LIN {X 0,Y 452.247,Z 648.153,A -85,B 0,C 180,E1 20026.851,E2 20026.851} C_VEL
LIN {X 0,Y 448.409,Z 632.212,A -85,B 0,C 180,E1 20025.069,E2 20025.069} C_VEL
LIN {X 0,Y 446.45,Z 614.687,A -85,B 0,C 180,E1 20023.26,E2 20023.26} C_VEL
LIN {X 0,Y 446.584,Z 593.795,A -85,B 0,C 180,E1 20021.279,E2 20021.279} C_VEL
LIN {X 0,Y 452.628,Z 538.562,A -85,B 0,C 180,E1 20016.48,E2 20016.48} C_VEL
LIN {X 0,Y 452.905,Z 536.236,A -85,B 0,C 180,E1 20016.274,E2 20016.274} C_VEL
LIN {X 0,Y 443.763,Z 516.786,A -85,B 0,C 180,E1 20013.042,E2 20013.042} C_VEL
LIN {X 0,Y 435.011,Z 498.685,A -85,B 0,C 180,E1 20009.766,E2 20009.766} C_VEL
LIN {X 0,Y 426.568,Z 481.843,A -85,B 0,C 180,E1 20006.443,E2 20006.443} C_VEL
LIN {X 0,Y 421.16,Z 471.659,A -85,B 0,C 180,E1 20004.249,E2 20004.249} C_VEL
LIN {X 0,Y 419.437,Z 467.925,A -85,B 0,C 180,E1 20003.459,E2 20003.459} C_VEL
LIN {X 0,Y 417.555,Z 464.51,A -85,B 0,C 180,E1 20002.676,E2 20002.676} C_VEL
LIN {X 0,Y 417.359,Z 463.499,A -85,B 0,C 180,E1 20002.464,E2 20002.464} C_VEL
LIN {X 0,Y 417.347,Z 463.499,A -85,B 0,C 180,E1 19998.431,E2 19998.431} C_VEL
LIN {X 0,Y 417.376,Z 463.496,A -85,B 0,C 180,E1 19994.579,E2 19994.579} C_VEL
LIN {X 0,Y 417.334,Z 463.503,A -85,B 0,C 180,E1 19990.63,E2 19990.63} C_VEL
LIN {X 0,Y 417.38,Z 463.495,A -85,B 0,C 180,E1 19986.741,E2 19986.741} C_VEL
LIN {X 0,Y 417.352,Z 463.498,A -85,B 0,C 180,E1 19982.884,E2 19982.884} C_VEL
LIN {X 0,Y 417.382,Z 463.493,A -85,B 0,C 180,E1 19979.039,E2 19979.039} C_VEL
LIN {X 0,Y 417.345,Z 463.498,A -85,B 0,C 180,E1 19975.19,E2 19975.19} C_VEL
LIN {X 0,Y 417.377,Z 463.478,A -85,B 0,C 180,E1 19971.458,E2 19971.458} C_VEL
LIN {X 0,Y 417.342,Z 463.486,A -85,B 0,C 180,E1 19967.688,E2 19967.688} C_VEL
LIN {X 0,Y 417.362,Z 463.495,A -85,B 0,C 180,E1 19963.579,E2 19963.579} C_VEL
LIN {X 0,Y 417.369,Z 463.498,A -85,B 0,C 180,E1 19959.82,E2 19959.82} C_VEL
LIN {X 0,Y 417.363,Z 463.495,A -85,B 0,C 180,E1 19955.886,E2 19955.886} C_VEL
LIN {X 0,Y 417.385,Z 463.489,A -85,B 0,C 180,E1 19951.996,E2 19951.996} C_VEL
LIN {X 0,Y 417.38,Z 463.491,A -85,B 0,C 180,E1 19947.997,E2 19947.997} C_VEL
LIN {X 0,Y 417.367,Z 463.496,A -85,B 0,C 180,E1 19944.23,E2 19944.23} C_VEL
LIN {X 0,Y 417.349,Z 463.5,A -85,B 0,C 180,E1 19940.266,E2 19940.266} C_VEL
LIN {X 0,Y 417.374,Z 463.49,A -85,B 0,C 180,E1 19936.54,E2 19936.54} C_VEL
LIN {X 0,Y 417.39,Z 463.643,A -85,B 0,C 180,E1 19936.338,E2 19936.338} C_VEL
LIN {X 0,Y 418.712,Z 467.029,A -85,B 0,C 180,E1 19935.791,E2 19935.791} C_VEL
LIN {X 0,Y 419.888,Z 469.412,A -85,B 0,C 180,E1 19935.374,E2 19935.374} C_VEL
LIN {X 0,Y 426.66,Z 483.707,A -85,B 0,C 180,E1 19932.995,E2 19932.995} C_VEL
LIN {X 0,Y 433.872,Z 500.582,A -85,B 0,C 180,E1 19930.525,E2 19930.525} C_VEL
LIN {X 0,Y 444.251,Z 519.272,A -85,B 0,C 180,E1 19928.996,E2 19928.996} C_VEL
LIN {X 0,Y 445.887,Z 529.867,A -85,B 0,C 180,E1 19928.609,E2 19928.609} C_VEL
LIN {X 0,Y 439.801,Z 761.275,A -85,B 0,C 180,E1 19924.551,E2 19924.551} C_VEL
LIN {X 0,Y 438.683,Z 782.005,A -85,B 0,C 180,E1 19923.967,E2 19923.967} C_VEL
LIN {X 0,Y 437.32,Z 800.081,A -85,B 0,C 180,E1 19923.255,E2 19923.255} C_VEL
LIN {X 0,Y 435.806,Z 807.622,A -85,B 0,C 180,E1 19922.975,E2 19922.975} C_VEL
LIN {X 0,Y 429.22,Z 824.782,A -85,B 0,C 180,E1 19922.434,E2 19922.434} C_VEL
LIN {X 0,Y 427.352,Z 831.771,A -85,B 0,C 180,E1 19922.067,E2 19922.067} C_VEL
LIN {X 0,Y 427.21,Z 832.734,A -85,B 0,C 180,E1 19922,E2 19922} C_VEL
LIN {X 0,Y 424.828,Z 850.823,A -85,B 0,C 180,E1 19920.624,E2 19920.624} C_VEL
LIN {X 0,Y 422.226,Z 868.674,A -85,B 0,C 180,E1 19918.964,E2 19918.964} C_VEL
LIN {X 0,Y 419.559,Z 885.444,A -85,B 0,C 180,E1 19917.075,E2 19917.075} C_VEL
LIN {X 0,Y 417.031,Z 900.766,A -85,B 0,C 180,E1 19915.003,E2 19915.003} C_VEL
LIN {X 0,Y 414.786,Z 914.246,A -85,B 0,C 180,E1 19912.835,E2 19912.835} C_VEL
LIN {X 0,Y 412.756,Z 926.896,A -85,B 0,C 180,E1 19910.415,E2 19910.415} C_VEL
LIN {X 0,Y 411.086,Z 938.068,A -85,B 0,C 180,E1 19907.845,E2 19907.845} C_VEL
LIN {X 0,Y 409.863,Z 947.306,A -85,B 0,C 180,E1 19905.275,E2 19905.275} C_VEL
LIN {X 0,Y 408.984,Z 955.199,A -85,B 0,C 180,E1 19902.566,E2 19902.566} C_VEL
LIN {X 0,Y 408.421,Z 961.6,A -85,B 0,C 180,E1 19899.724,E2 19899.724} C_VEL
LIN {X 0,Y 408.141,Z 966.263,A -85,B 0,C 180,E1 19896.894,E2 19896.894} C_VEL
LIN {X 0,Y 408.022,Z 969.312,A -85,B 0,C 180,E1 19894.074,E2 19894.074} C_VEL
LIN {X 0,Y 407.98,Z 970.823,A -85,B 0,C 180,E1 19891.263,E2 19891.263} C_VEL
LIN {X 0,Y 407.98,Z 970.794,A -85,B 0,C 180,E1 19888.454,E2 19888.454} C_VEL
LIN {X 0,Y 408.024,Z 969.165,A -85,B 0,C 180,E1 19885.643,E2 19885.643} C_VEL
LIN {X 0,Y 408.152,Z 965.977,A -85,B 0,C 180,E1 19882.812,E2 19882.812} C_VEL
LIN {X 0,Y 408.449,Z 961.195,A -85,B 0,C 180,E1 19879.99,E2 19879.99} C_VEL
LIN {X 0,Y 409.002,Z 954.992,A -85,B 0,C 180,E1 19877.268,E2 19877.268} C_VEL
LIN {X 0,Y 409.947,Z 946.693,A -85,B 0,C 180,E1 19874.437,E2 19874.437} C_VEL
LIN {X 0,Y 411.285,Z 936.743,A -85,B 0,C 180,E1 19871.723,E2 19871.723} C_VEL
LIN {X 0,Y 412.905,Z 925.95,A -85,B 0,C 180,E1 19869.295,E2 19869.295} C_VEL
LIN {X 0,Y 414.977,Z 913.101,A -85,B 0,C 180,E1 19866.874,E2 19866.874} C_VEL
LIN {X 0,Y 417.417,Z 898.384,A -85,B 0,C 180,E1 19864.562,E2 19864.562} C_VEL
LIN {X 0,Y 420.016,Z 882.599,A -85,B 0,C 180,E1 19862.494,E2 19862.494} C_VEL
LIN {X 0,Y 422.519,Z 866.692,A -85,B 0,C 180,E1 19860.746,E2 19860.746} C_VEL
LIN {X 0,Y 425.074,Z 849.262,A -85,B 0,C 180,E1 19859.15,E2 19859.15} C_VEL
LIN {X 0,Y 427.469,Z 830.816,A -85,B 0,C 180,E1 19857.771,E2 19857.771} C_VEL
LIN {X 0,Y 429.58,Z 811.902,A -85,B 0,C 180,E1 19856.637,E2 19856.637} C_VEL
LIN {X 0,Y 431.357,Z 792.246,A -85,B 0,C 180,E1 19855.718,E2 19855.718} C_VEL
LIN {X 0,Y 432.78,Z 770.977,A -85,B 0,C 180,E1 19854.992,E2 19854.992} C_VEL
LIN {X 0,Y 433.737,Z 747.508,A -85,B 0,C 180,E1 19854.477,E2 19854.477} C_VEL
LIN {X 0,Y 439.275,Z 540.89,A -85,B 0,C 180,E1 19850.824,E2 19850.824} C_VEL
LIN {X 0,Y 433.898,Z 520.693,A -85,B 0,C 180,E1 19849.809,E2 19849.809} C_VEL
LIN {X 0,Y 423.787,Z 502.841,A -85,B 0,C 180,E1 19848.207,E2 19848.207} C_VEL
LIN {X 0,Y 418.624,Z 487.868,A -85,B 0,C 180,E1 19845.378,E2 19845.378} C_VEL
LIN {X 0,Y 413.554,Z 474.797,A -85,B 0,C 180,E1 19842.607,E2 19842.607} C_VEL
LIN {X 0,Y 410.381,Z 467.367,A -85,B 0,C 180,E1 19840.948,E2 19840.948} C_VEL
LIN {X 0,Y 410.03,Z 466.658,A -85,B 0,C 180,E1 19840.761,E2 19840.761} C_VEL
LIN {X 0,Y 415.308,Z 479.497,A -85,B 0,C 180,E1 19838.4,E2 19838.4} C_VEL
LIN {X 0,Y 422.076,Z 497.495,A -85,B 0,C 180,E1 19835.311,E2 19835.311} C_VEL
LIN {X 0,Y 428.337,Z 516.103,A -85,B 0,C 180,E1 19832.349,E2 19832.349} C_VEL
LIN {X 0,Y 425.447,Z 549.874,A -85,B 0,C 180,E1 19828.572,E2 19828.572} C_VEL
LIN {X 0,Y 422.614,Z 585.893,A -85,B 0,C 180,E1 19824.608,E2 19824.608} C_VEL
LIN {X 0,Y 420.128,Z 621.951,A -85,B 0,C 180,E1 19820.731,E2 19820.731} C_VEL
LIN {X 0,Y 420.828,Z 628.627,A -85,B 0,C 180,E1 19820.519,E2 19820.519} C_VEL
LIN {X 0,Y 416.374,Z 763.577,A -85,B 0,C 180,E1 19817.315,E2 19817.315} C_VEL
LIN {X 0,Y 415.988,Z 779.751,A -85,B 0,C 180,E1 19816.715,E2 19816.715} C_VEL
LIN {X 0,Y 415.353,Z 795.906,A -85,B 0,C 180,E1 19815.856,E2 19815.856} C_VEL
LIN {X 0,Y 414.592,Z 810.59,A -85,B 0,C 180,E1 19814.812,E2 19814.812} C_VEL
LIN {X 0,Y 413.68,Z 825.181,A -85,B 0,C 180,E1 19813.488,E2 19813.488} C_VEL
LIN {X 0,Y 412.722,Z 838.536,A -85,B 0,C 180,E1 19811.955,E2 19811.955} C_VEL
LIN {X 0,Y 411.812,Z 850.761,A -85,B 0,C 180,E1 19810.209,E2 19810.209} C_VEL
LIN {X 0,Y 410.995,Z 861.622,A -85,B 0,C 180,E1 19808.253,E2 19808.253} C_VEL
LIN {X 0,Y 410.392,Z 870.255,A -85,B 0,C 180,E1 19806.295,E2 19806.295} C_VEL
LIN {X 0,Y 409.918,Z 877.846,A -85,B 0,C 180,E1 19804.056,E2 19804.056} C_VEL
LIN {X 0,Y 409.653,Z 883.079,A -85,B 0,C 180,E1 19801.958,E2 19801.958} C_VEL
LIN {X 0,Y 409.548,Z 887.055,A -85,B 0,C 180,E1 19799.581,E2 19799.581} C_VEL
LIN {X 0,Y 409.583,Z 888.99,A -85,B 0,C 180,E1 19797.342,E2 19797.342} C_VEL
LIN {X 0,Y 409.775,Z 889.229,A -85,B 0,C 180,E1 19794.961,E2 19794.961} C_VEL
LIN {X 0,Y 410.11,Z 887.636,A -85,B 0,C 180,E1 19792.717,E2 19792.717} C_VEL
LIN {X 0,Y 410.655,Z 884.296,A -85,B 0,C 180,E1 19790.437,E2 19790.437} C_VEL
LIN {X 0,Y 411.479,Z 878.755,A -85,B 0,C 180,E1 19788.08,E2 19788.08} C_VEL
LIN {X 0,Y 412.372,Z 872.331,A -85,B 0,C 180,E1 19786.111,E2 19786.111} C_VEL
LIN {X 0,Y 413.597,Z 863.352,A -85,B 0,C 180,E1 19784.003,E2 19784.003} C_VEL
LIN {X 0,Y 414.895,Z 853.205,A -85,B 0,C 180,E1 19782.162,E2 19782.162} C_VEL
LIN {X 0,Y 416.186,Z 842.184,A -85,B 0,C 180,E1 19780.565,E2 19780.565} C_VEL
LIN {X 0,Y 417.51,Z 829.221,A -85,B 0,C 180,E1 19779.065,E2 19779.065} C_VEL
LIN {X 0,Y 418.633,Z 815.574,A -85,B 0,C 180,E1 19777.83,E2 19777.83} C_VEL
LIN {X 0,Y 419.575,Z 800.482,A -85,B 0,C 180,E1 19776.772,E2 19776.772} C_VEL
LIN {X 0,Y 420.221,Z 784.494,A -85,B 0,C 180,E1 19775.954,E2 19775.954} C_VEL
LIN {X 0,Y 421.597,Z 753.425,A -85,B 0,C 180,E1 19774.815,E2 19774.815} C_VEL
LIN {X 0,Y 431.426,Z 657.119,A -85,B 0,C 180,E1 19771.483,E2 19771.483} C_VEL
LIN {X 0,Y 438.558,Z 643.152,A -85,B 0,C 180,E1 19770.302,E2 19770.302} C_VEL
LIN {X 0,Y 445.715,Z 621.577,A -85,B 0,C 180,E1 19767.121,E2 19767.121} C_VEL
LIN {X 0,Y 453.266,Z 605.107,A -85,B 0,C 180,E1 19764.487,E2 19764.487} C_VEL
LIN {X 0,Y 461.57,Z 591.773,A -85,B 0,C 180,E1 19762.171,E2 19762.171} C_VEL
LIN {X 0,Y 453.703,Z 603.277,A -85,B 0,C 180,E1 19760.474,E2 19760.474} C_VEL
LIN {X 0,Y 447.749,Z 615.574,A -85,B 0,C 180,E1 19758.619,E2 19758.619} C_VEL
LIN {X 0,Y 444.305,Z 627.955,A -85,B 0,C 180,E1 19756.711,E2 19756.711} C_VEL
LIN {X 0,Y 443.385,Z 639.929,A -85,B 0,C 180,E1 19754.838,E2 19754.838} C_VEL
LIN {X 0,Y 444.836,Z 652.133,A -85,B 0,C 180,E1 19752.927,E2 19752.927} C_VEL
LIN {X 0,Y 448.588,Z 663.737,A -85,B 0,C 180,E1 19751.112,E2 19751.112} C_VEL
LIN {X 0,Y 454.843,Z 675.364,A -85,B 0,C 180,E1 19749.305,E2 19749.305} C_VEL
LIN {X 0,Y 461.889,Z 684.775,A -85,B 0,C 180,E1 19747.858,E2 19747.858} C_VEL
LIN {X 0,Y 450.972,Z 703.36,A -85,B 0,C 180,E1 19747.17,E2 19747.17} C_VEL
LIN {X 0,Y 442.545,Z 720.539,A -85,B 0,C 180,E1 19746.376,E2 19746.376} C_VEL
LIN {X 0,Y 438.274,Z 731,A -85,B 0,C 180,E1 19745.853,E2 19745.853} C_VEL
LIN {X 0,Y 435.008,Z 751.2,A -85,B 0,C 180,E1 19745.76,E2 19745.76} C_VEL
LIN {X 0,Y 432.722,Z 773.487,A -85,B 0,C 180,E1 19745.533,E2 19745.533} C_VEL
LIN {X 0,Y 431.639,Z 803.634,A -85,B 0,C 180,E1 19744.962,E2 19744.962} C_VEL
LIN {X 0,Y 430.206,Z 824.359,A -85,B 0,C 180,E1 19744.347,E2 19744.347} C_VEL
LIN {X 0,Y 428.359,Z 844.316,A -85,B 0,C 180,E1 19743.507,E2 19743.507} C_VEL
LIN {X 0,Y 426.167,Z 863.94,A -85,B 0,C 180,E1 19742.419,E2 19742.419} C_VEL
LIN {X 0,Y 423.795,Z 882.686,A -85,B 0,C 180,E1 19741.111,E2 19741.111} C_VEL
LIN {X 0,Y 421.195,Z 901.021,A -85,B 0,C 180,E1 19739.546,E2 19739.546} C_VEL
LIN {X 0,Y 418.667,Z 918.311,A -85,B 0,C 180,E1 19737.756,E2 19737.756} C_VEL
LIN {X 0,Y 416.222,Z 934.359,A -85,B 0,C 180,E1 19735.774,E2 19735.774} C_VEL
LIN {X 0,Y 414.071,Z 948.963,A -85,B 0,C 180,E1 19733.632,E2 19733.632} C_VEL
LIN {X 0,Y 412.098,Z 962.898,A -85,B 0,C 180,E1 19731.194,E2 19731.194} C_VEL
LIN {X 0,Y 410.508,Z 975.21,A -85,B 0,C 180,E1 19728.608,E2 19728.608} C_VEL
LIN {X 0,Y 409.439,Z 985.412,A -85,B 0,C 180,E1 19726.019,E2 19726.019} C_VEL
LIN {X 0,Y 408.7,Z 994.21,A -85,B 0,C 180,E1 19723.296,E2 19723.296} C_VEL
LIN {X 0,Y 408.279,Z 1001.508,A -85,B 0,C 180,E1 19720.442,E2 19720.442} C_VEL
LIN {X 0,Y 408.135,Z 1006.746,A -85,B 0,C 180,E1 19717.744,E2 19717.744} C_VEL
LIN {X 0,Y 408.111,Z 1010.345,A -85,B 0,C 180,E1 19715.061,E2 19715.061} C_VEL
LIN {X 0,Y 408.146,Z 1012.401,A -85,B 0,C 180,E1 19712.388,E2 19712.388} C_VEL
LIN {X 0,Y 408.157,Z 1012.992,A -85,B 0,C 180,E1 19709.58,E2 19709.58} C_VEL
LIN {X 0,Y 408.13,Z 1012.047,A -85,B 0,C 180,E1 19706.911,E2 19706.911} C_VEL
LIN {X 0,Y 408.1,Z 1009.523,A -85,B 0,C 180,E1 19704.236,E2 19704.236} C_VEL
LIN {X 0,Y 408.152,Z 1005.246,A -85,B 0,C 180,E1 19701.407,E2 19701.407} C_VEL
LIN {X 0,Y 408.354,Z 999.555,A -85,B 0,C 180,E1 19698.705,E2 19698.705} C_VEL
LIN {X 0,Y 408.82,Z 992.138,A -85,B 0,C 180,E1 19695.989,E2 19695.989} C_VEL
LIN {X 0,Y 409.665,Z 982.783,A -85,B 0,C 180,E1 19693.263,E2 19693.263} C_VEL
LIN {X 0,Y 410.881,Z 971.974,A -85,B 0,C 180,E1 19690.674,E2 19690.674} C_VEL
LIN {X 0,Y 412.492,Z 959.502,A -85,B 0,C 180,E1 19688.182,E2 19688.182} C_VEL
LIN {X 0,Y 414.56,Z 945.232,A -85,B 0,C 180,E1 19685.795,E2 19685.795} C_VEL
LIN {X 0,Y 416.83,Z 930.021,A -85,B 0,C 180,E1 19683.657,E2 19683.657} C_VEL
LIN {X 0,Y 419.242,Z 914.205,A -85,B 0,C 180,E1 19681.782,E2 19681.782} C_VEL
LIN {X 0,Y 421.803,Z 896.64,A -85,B 0,C 180,E1 19680.042,E2 19680.042} C_VEL
LIN {X 0,Y 424.332,Z 878.099,A -85,B 0,C 180,E1 19678.537,E2 19678.537} C_VEL
LIN {X 0,Y 426.655,Z 859.244,A -85,B 0,C 180,E1 19677.297,E2 19677.297} C_VEL
LIN {X 0,Y 428.718,Z 839.82,A -85,B 0,C 180,E1 19676.286,E2 19676.286} C_VEL
LIN {X 0,Y 430.514,Z 819.136,A -85,B 0,C 180,E1 19675.477,E2 19675.477} C_VEL
LIN {X 0,Y 431.819,Z 798.409,A -85,B 0,C 180,E1 19674.917,E2 19674.917} C_VEL
LIN {X 0,Y 432.958,Z 768.448,A -85,B 0,C 180,E1 19674.395,E2 19674.395} C_VEL
LIN {X 0,Y 434.942,Z 748.992,A -85,B 0,C 180,E1 19674.194,E2 19674.194} C_VEL
LIN {X 0,Y 448.015,Z 719.06,A -85,B 0,C 180,E1 19672.608,E2 19672.608} C_VEL
LIN {X 0,Y 457.258,Z 701.76,A -85,B 0,C 180,E1 19671.851,E2 19671.851} C_VEL
LIN {X 0,Y 465.342,Z 688.644,A -85,B 0,C 180,E1 19671.376,E2 19671.376} C_VEL
LIN {X 0,Y 456.514,Z 676.324,A -85,B 0,C 180,E1 19669.657,E2 19669.657} C_VEL
LIN {X 0,Y 449.449,Z 662.719,A -85,B 0,C 180,E1 19667.895,E2 19667.895} C_VEL
LIN {X 0,Y 444.221,Z 647.515,A -85,B 0,C 180,E1 19666.076,E2 19666.076} C_VEL
LIN {X 0,Y 440.778,Z 630.005,A -85,B 0,C 180,E1 19664.138,E2 19664.138} C_VEL
LIN {X 0,Y 439.519,Z 612.252,A -85,B 0,C 180,E1 19662.326,E2 19662.326} C_VEL
LIN {X 0,Y 440.316,Z 590.385,A -85,B 0,C 180,E1 19660.273,E2 19660.273} C_VEL
LIN {X 0,Y 445.999,Z 543.065,A -85,B 0,C 180,E1 19656.129,E2 19656.129} C_VEL
LIN {X 0,Y 446.371,Z 539.996,A -85,B 0,C 180,E1 19655.856,E2 19655.856} C_VEL
LIN {X 0,Y 436.422,Z 518.757,A -85,B 0,C 180,E1 19652.263,E2 19652.263} C_VEL
LIN {X 0,Y 427.384,Z 500.161,A -85,B 0,C 180,E1 19648.812,E2 19648.812} C_VEL
LIN {X 0,Y 418.385,Z 482.388,A -85,B 0,C 180,E1 19645.175,E2 19645.175} C_VEL
LIN {X 0,Y 413.379,Z 472.882,A -85,B 0,C 180,E1 19643.069,E2 19643.069} C_VEL
LIN {X 0,Y 411.325,Z 468.748,A -85,B 0,C 180,E1 19642.134,E2 19642.134} C_VEL
LIN {X 0,Y 409.559,Z 465.216,A -85,B 0,C 180,E1 19641.331,E2 19641.331} C_VEL
LIN {X 0,Y 409.423,Z 464.486,A -85,B 0,C 180,E1 19641.188,E2 19641.188} C_VEL
LIN {X 0,Y 409.427,Z 464.488,A -85,B 0,C 180,E1 19637.187,E2 19637.187} C_VEL
LIN {X 0,Y 409.442,Z 464.486,A -85,B 0,C 180,E1 19633.414,E2 19633.414} C_VEL
LIN {X 0,Y 409.438,Z 464.484,A -85,B 0,C 180,E1 19629.275,E2 19629.275} C_VEL
LIN {X 0,Y 409.427,Z 464.486,A -85,B 0,C 180,E1 19625.465,E2 19625.465} C_VEL
LIN {X 0,Y 409.435,Z 464.485,A -85,B 0,C 180,E1 19621.399,E2 19621.399} C_VEL
LIN {X 0,Y 409.423,Z 464.487,A -85,B 0,C 180,E1 19617.62,E2 19617.62} C_VEL
LIN {X 0,Y 409.404,Z 464.481,A -85,B 0,C 180,E1 19613.549,E2 19613.549} C_VEL
LIN {X 0,Y 409.434,Z 464.486,A -85,B 0,C 180,E1 19609.731,E2 19609.731} C_VEL
LIN {X 0,Y 409.393,Z 464.479,A -85,B 0,C 180,E1 19605.831,E2 19605.831} C_VEL
LIN {X 0,Y 409.437,Z 464.466,A -85,B 0,C 180,E1 19601.932,E2 19601.932} C_VEL
LIN {X 0,Y 409.419,Z 464.473,A -85,B 0,C 180,E1 19598.059,E2 19598.059} C_VEL
LIN {X 0,Y 409.442,Z 464.481,A -85,B 0,C 180,E1 19594.235,E2 19594.235} C_VEL
LIN {X 0,Y 409.413,Z 464.489,A -85,B 0,C 180,E1 19590.389,E2 19590.389} C_VEL
LIN {X 0,Y 409.442,Z 464.483,A -85,B 0,C 180,E1 19586.503,E2 19586.503} C_VEL
LIN {X 0,Y 409.404,Z 464.483,A -85,B 0,C 180,E1 19582.722,E2 19582.722} C_VEL
LIN {X 0,Y 409.416,Z 464.478,A -85,B 0,C 180,E1 19578.747,E2 19578.747} C_VEL
LIN {X 0,Y 409.454,Z 464.596,A -85,B 0,C 180,E1 19577.399,E2 19577.399} C_VEL
LIN {X 0,Y 410.728,Z 467.94,A -85,B 0,C 180,E1 19576.838,E2 19576.838} C_VEL
LIN {X 0,Y 411.906,Z 470.18,A -85,B 0,C 180,E1 19576.419,E2 19576.419} C_VEL
LIN {X 0,Y 418.963,Z 484.85,A -85,B 0,C 180,E1 19573.885,E2 19573.885} C_VEL
LIN {X 0,Y 426.18,Z 501.197,A -85,B 0,C 180,E1 19571.41,E2 19571.41} C_VEL
LIN {X 0,Y 438.347,Z 522.672,A -85,B 0,C 180,E1 19569.559,E2 19569.559} C_VEL
LIN {X 0,Y 439.628,Z 531.441,A -85,B 0,C 180,E1 19569.237,E2 19569.237} C_VEL
LIN {X 0,Y 433.238,Z 761.59,A -85,B 0,C 180,E1 19565.151,E2 19565.151} C_VEL
LIN {X 0,Y 432.073,Z 782.349,A -85,B 0,C 180,E1 19564.56,E2 19564.56} C_VEL
LIN {X 0,Y 430.416,Z 802.881,A -85,B 0,C 180,E1 19563.724,E2 19563.724} C_VEL
LIN {X 0,Y 428.44,Z 822.386,A -85,B 0,C 180,E1 19562.671,E2 19562.671} C_VEL
LIN {X 0,Y 427.21,Z 832.734,A -85,B 0,C 180,E1 19562,E2 19562} C_VEL
LIN {X 0,Y 425.5,Z 839.763,A -85,B 0,C 180,E1 19561.577,E2 19561.577} C_VEL
LIN {X 0,Y 417.937,Z 856.908,A -85,B 0,C 180,E1 19560.609,E2 19560.609} C_VEL
LIN {X 0,Y 416.078,Z 863.292,A -85,B 0,C 180,E1 19560.078,E2 19560.078} C_VEL
LIN {X 0,Y 413.363,Z 879.928,A -85,B 0,C 180,E1 19558.299,E2 19558.299} C_VEL
LIN {X 0,Y 410.686,Z 895.548,A -85,B 0,C 180,E1 19556.301,E2 19556.301} C_VEL
LIN {X 0,Y 408.214,Z 909.683,A -85,B 0,C 180,E1 19554.144,E2 19554.144} C_VEL
LIN {X 0,Y 405.949,Z 922.609,A -85,B 0,C 180,E1 19551.788,E2 19551.788} C_VEL
LIN {X 0,Y 404.098,Z 933.776,A -85,B 0,C 180,E1 19549.362,E2 19549.362} C_VEL
LIN {X 0,Y 402.506,Z 944.324,A -85,B 0,C 180,E1 19546.598,E2 19546.598} C_VEL
LIN {X 0,Y 401.402,Z 952.875,A -85,B 0,C 180,E1 19543.834,E2 19543.834} C_VEL
LIN {X 0,Y 400.688,Z 959.675,A -85,B 0,C 180,E1 19541.077,E2 19541.077} C_VEL
LIN {X 0,Y 400.274,Z 965.045,A -85,B 0,C 180,E1 19538.185,E2 19538.185} C_VEL
LIN {X 0,Y 400.068,Z 968.705,A -85,B 0,C 180,E1 19535.305,E2 19535.305} C_VEL
LIN {X 0,Y 400.006,Z 970.799,A -85,B 0,C 180,E1 19532.435,E2 19532.435} C_VEL
LIN {X 0,Y 399.991,Z 971.379,A -85,B 0,C 180,E1 19529.57,E2 19529.57} C_VEL
LIN {X 0,Y 400.015,Z 970.445,A -85,B 0,C 180,E1 19526.704,E2 19526.704} C_VEL
LIN {X 0,Y 400.115,Z 967.88,A -85,B 0,C 180,E1 19523.831,E2 19523.831} C_VEL
LIN {X 0,Y 400.362,Z 963.724,A -85,B 0,C 180,E1 19520.947,E2 19520.947} C_VEL
LIN {X 0,Y 400.847,Z 957.884,A -85,B 0,C 180,E1 19518.051,E2 19518.051} C_VEL
LIN {X 0,Y 401.675,Z 950.656,A -85,B 0,C 180,E1 19515.291,E2 19515.291} C_VEL
LIN {X 0,Y 402.918,Z 941.604,A -85,B 0,C 180,E1 19512.526,E2 19512.526} C_VEL
LIN {X 0,Y 404.663,Z 930.439,A -85,B 0,C 180,E1 19509.761,E2 19509.761} C_VEL
LIN {X 0,Y 406.836,Z 917.595,A -85,B 0,C 180,E1 19507.15,E2 19507.15} C_VEL
LIN {X 0,Y 409.221,Z 903.913,A -85,B 0,C 180,E1 19504.84,E2 19504.84} C_VEL
LIN {X 0,Y 411.772,Z 889.246,A -85,B 0,C 180,E1 19502.76,E2 19502.76} C_VEL
LIN {X 0,Y 414.527,Z 873.003,A -85,B 0,C 180,E1 19500.828,E2 19500.828} C_VEL
LIN {X 0,Y 417.337,Z 855.065,A -85,B 0,C 180,E1 19499.06,E2 19499.06} C_VEL
LIN {X 0,Y 419.924,Z 837.057,A -85,B 0,C 180,E1 19497.605,E2 19497.605} C_VEL
LIN {X 0,Y 422.208,Z 818.712,A -85,B 0,C 180,E1 19496.398,E2 19496.398} C_VEL
LIN {X 0,Y 424.212,Z 799.183,A -85,B 0,C 180,E1 19495.386,E2 19495.386} C_VEL
LIN {X 0,Y 425.793,Z 779.188,A -85,B 0,C 180,E1 19494.615,E2 19494.615} C_VEL
LIN {X 0,Y 426.869,Z 758.771,A -85,B 0,C 180,E1 19494.067,E2 19494.067} C_VEL
LIN {X 0,Y 433.03,Z 542.633,A -85,B 0,C 180,E1 19490.18,E2 19490.18} C_VEL
LIN {X 0,Y 428.346,Z 524.911,A -85,B 0,C 180,E1 19489.267,E2 19489.267} C_VEL
LIN {X 0,Y 417.742,Z 506.393,A -85,B 0,C 180,E1 19487.569,E2 19487.569} C_VEL
LIN {X 0,Y 416.036,Z 503.201,A -85,B 0,C 180,E1 19487.241,E2 19487.241} C_VEL
LIN {X 0,Y 410.685,Z 488.339,A -85,B 0,C 180,E1 19484.326,E2 19484.326} C_VEL
LIN {X 0,Y 405.937,Z 476.291,A -85,B 0,C 180,E1 19481.685,E2 19481.685} C_VEL
LIN {X 0,Y 404.161,Z 472.316,A -85,B 0,C 180,E1 19480.738,E2 19480.738} C_VEL
LIN {X 0,Y 411.069,Z 489.811,A -85,B 0,C 180,E1 19477.537,E2 19477.537} C_VEL
LIN {X 0,Y 417.829,Z 508.675,A -85,B 0,C 180,E1 19474.351,E2 19474.351} C_VEL
LIN {X 0,Y 421.262,Z 519.171,A -85,B 0,C 180,E1 19472.682,E2 19472.682} C_VEL
LIN {X 0,Y 418.161,Z 553.481,A -85,B 0,C 180,E1 19468.804,E2 19468.804} C_VEL
LIN {X 0,Y 415.231,Z 589.559,A -85,B 0,C 180,E1 19464.795,E2 19464.795} C_VEL
LIN {X 0,Y 412.862,Z 623.388,A -85,B 0,C 180,E1 19461.15,E2 19461.15} C_VEL
LIN {X 0,Y 413.48,Z 629.666,A -85,B 0,C 180,E1 19460.943,E2 19460.943} C_VEL
LIN {X 0,Y 408.78,Z 764.001,A -85,B 0,C 180,E1 19457.659,E2 19457.659} C_VEL
LIN {X 0,Y 408.388,Z 780.031,A -85,B 0,C 180,E1 19457.062,E2 19457.062} C_VEL
LIN {X 0,Y 407.703,Z 796.723,A -85,B 0,C 180,E1 19456.162,E2 19456.162} C_VEL
LIN {X 0,Y 406.907,Z 811.445,A -85,B 0,C 180,E1 19455.098,E2 19455.098} C_VEL
LIN {X 0,Y 405.936,Z 826.289,A -85,B 0,C 180,E1 19453.727,E2 19453.727} C_VEL
LIN {X 0,Y 404.953,Z 839.471,A -85,B 0,C 180,E1 19452.187,E2 19452.187} C_VEL
LIN {X 0,Y 404.002,Z 851.751,A -85,B 0,C 180,E1 19450.409,E2 19450.409} C_VEL
LIN {X 0,Y 403.146,Z 862.656,A -85,B 0,C 180,E1 19448.414,E2 19448.414} C_VEL
LIN {X 0,Y 402.516,Z 871.354,A -85,B 0,C 180,E1 19446.418,E2 19446.418} C_VEL
LIN {X 0,Y 402.022,Z 879.004,A -85,B 0,C 180,E1 19444.136,E2 19444.136} C_VEL
LIN {X 0,Y 401.749,Z 884.296,A -85,B 0,C 180,E1 19441.997,E2 19441.997} C_VEL
LIN {X 0,Y 401.644,Z 888.328,A -85,B 0,C 180,E1 19439.572,E2 19439.572} C_VEL
LIN {X 0,Y 401.692,Z 890.316,A -85,B 0,C 180,E1 19437.29,E2 19437.29} C_VEL
LIN {X 0,Y 401.909,Z 890.606,A -85,B 0,C 180,E1 19434.862,E2 19434.862} C_VEL
LIN {X 0,Y 402.286,Z 889.071,A -85,B 0,C 180,E1 19432.574,E2 19432.574} C_VEL
LIN {X 0,Y 402.877,Z 885.858,A -85,B 0,C 180,E1 19430.284,E2 19430.284} C_VEL
LIN {X 0,Y 403.719,Z 880.679,A -85,B 0,C 180,E1 19427.993,E2 19427.993} C_VEL
LIN {X 0,Y 404.763,Z 873.969,A -85,B 0,C 180,E1 19425.845,E2 19425.845} C_VEL
LIN {X 0,Y 405.994,Z 865.73,A -85,B 0,C 180,E1 19423.839,E2 19423.839} C_VEL
LIN {X 0,Y 407.358,Z 855.976,A -85,B 0,C 180,E1 19421.985,E2 19421.985} C_VEL
LIN {X 0,Y 408.83,Z 844.758,A -85,B 0,C 180,E1 19420.276,E2 19420.276} C_VEL
LIN {X 0,Y 410.28,Z 831.662,A -85,B 0,C 180,E1 19418.709,E2 19418.709} C_VEL
LIN {X 0,Y 411.54,Z 818.132,A -85,B 0,C 180,E1 19417.427,E2 19417.427} C_VEL
LIN {X 0,Y 412.561,Z 803.674,A -85,B 0,C 180,E1 19416.364,E2 19416.364} C_VEL
LIN {X 0,Y 413.348,Z 787.167,A -85,B 0,C 180,E1 19415.47,E2 19415.47} C_VEL
LIN {X 0,Y 414.903,Z 756.833,A -85,B 0,C 180,E1 19414.279,E2 19414.279} C_VEL
LIN {X 0,Y 425.848,Z 660.115,A -85,B 0,C 180,E1 19410.767,E2 19410.767} C_VEL
LIN {X 0,Y 433.367,Z 645.952,A -85,B 0,C 180,E1 19409.574,E2 19409.574} C_VEL
LIN {X 0,Y 441.041,Z 625.163,A -85,B 0,C 180,E1 19406.416,E2 19406.416} C_VEL
LIN {X 0,Y 449.009,Z 609.528,A -85,B 0,C 180,E1 19403.836,E2 19403.836} C_VEL
LIN {X 0,Y 454.853,Z 600.657,A -85,B 0,C 180,E1 19402.236,E2 19402.236} C_VEL
LIN {X 0,Y 447.156,Z 612.063,A -85,B 0,C 180,E1 19400.484,E2 19400.484} C_VEL
LIN {X 0,Y 441.777,Z 623.28,A -85,B 0,C 180,E1 19398.713,E2 19398.713} C_VEL
LIN {X 0,Y 438.509,Z 635.367,A -85,B 0,C 180,E1 19396.762,E2 19396.762} C_VEL
LIN {X 0,Y 437.725,Z 647.141,A -85,B 0,C 180,E1 19394.836,E2 19394.836} C_VEL
LIN {X 0,Y 439.408,Z 659.195,A -85,B 0,C 180,E1 19392.873,E2 19392.873} C_VEL
LIN {X 0,Y 443.526,Z 670.976,A -85,B 0,C 180,E1 19390.957,E2 19390.957} C_VEL
LIN {X 0,Y 449.983,Z 682.329,A -85,B 0,C 180,E1 19389.128,E2 19389.128} C_VEL
LIN {X 0,Y 453.361,Z 687.303,A -85,B 0,C 180,E1 19388.364,E2 19388.364} C_VEL
LIN {X 0,Y 442.963,Z 705.582,A -85,B 0,C 180,E1 19387.656,E2 19387.656} C_VEL
LIN {X 0,Y 434.5,Z 723.436,A -85,B 0,C 180,E1 19386.793,E2 19386.793} C_VEL
LIN {X 0,Y 431.94,Z 729.896,A -85,B 0,C 180,E1 19386.48,E2 19386.48} C_VEL
LIN {X 0,Y 428.586,Z 750.592,A -85,B 0,C 180,E1 19386.389,E2 19386.389} C_VEL
LIN {X 0,Y 426.227,Z 773.378,A -85,B 0,C 180,E1 19386.156,E2 19386.156} C_VEL
LIN {X 0,Y 425.101,Z 803.073,A -85,B 0,C 180,E1 19385.589,E2 19385.589} C_VEL
LIN {X 0,Y 423.59,Z 823.902,A -85,B 0,C 180,E1 19384.965,E2 19384.965} C_VEL
LIN {X 0,Y 421.647,Z 843.95,A -85,B 0,C 180,E1 19384.113,E2 19384.113} C_VEL
LIN {X 0,Y 419.478,Z 862.427,A -85,B 0,C 180,E1 19383.083,E2 19383.083} C_VEL
LIN {X 0,Y 416.921,Z 881.674,A -85,B 0,C 180,E1 19381.738,E2 19381.738} C_VEL
LIN {X 0,Y 414.159,Z 900.216,A -85,B 0,C 180,E1 19380.143,E2 19380.143} C_VEL
LIN {X 0,Y 411.522,Z 917.291,A -85,B 0,C 180,E1 19378.36,E2 19378.36} C_VEL
LIN {X 0,Y 408.908,Z 933.434,A -85,B 0,C 180,E1 19376.348,E2 19376.348} C_VEL
LIN {X 0,Y 406.535,Z 948.549,A -85,B 0,C 180,E1 19374.097,E2 19374.097} C_VEL
LIN {X 0,Y 404.412,Z 962.481,A -85,B 0,C 180,E1 19371.617,E2 19371.617} C_VEL
LIN {X 0,Y 402.719,Z 974.792,A -85,B 0,C 180,E1 19368.981,E2 19368.981} C_VEL
LIN {X 0,Y 401.566,Z 984.994,A -85,B 0,C 180,E1 19366.342,E2 19366.342} C_VEL
LIN {X 0,Y 400.748,Z 993.792,A -85,B 0,C 180,E1 19363.565,E2 19363.565} C_VEL
LIN {X 0,Y 400.3,Z 1001.092,A -85,B 0,C 180,E1 19360.652,E2 19360.652} C_VEL
LIN {X 0,Y 400.15,Z 1006.332,A -85,B 0,C 180,E1 19357.9,E2 19357.9} C_VEL
LIN {X 0,Y 400.112,Z 1009.932,A -85,B 0,C 180,E1 19355.162,E2 19355.162} C_VEL
LIN {X 0,Y 400.154,Z 1011.989,A -85,B 0,C 180,E1 19352.435,E2 19352.435} C_VEL
LIN {X 0,Y 400.168,Z 1012.581,A -85,B 0,C 180,E1 19349.571,E2 19349.571} C_VEL
LIN {X 0,Y 400.138,Z 1011.635,A -85,B 0,C 180,E1 19346.849,E2 19346.849} C_VEL
LIN {X 0,Y 400.107,Z 1009.014,A -85,B 0,C 180,E1 19344.037,E2 19344.037} C_VEL
LIN {X 0,Y 400.154,Z 1004.83,A -85,B 0,C 180,E1 19341.234,E2 19341.234} C_VEL
LIN {X 0,Y 400.383,Z 999.137,A -85,B 0,C 180,E1 19338.477,E2 19338.477} C_VEL
LIN {X 0,Y 400.889,Z 991.718,A -85,B 0,C 180,E1 19335.706,E2 19335.706} C_VEL
LIN {X 0,Y 401.796,Z 982.362,A -85,B 0,C 180,E1 19332.925,E2 19332.925} C_VEL
LIN {X 0,Y 403.123,Z 971.553,A -85,B 0,C 180,E1 19330.287,E2 19330.287} C_VEL
LIN {X 0,Y 404.809,Z 959.344,A -85,B 0,C 180,E1 19327.797,E2 19327.797} C_VEL
LIN {X 0,Y 407.008,Z 945.075,A -85,B 0,C 180,E1 19325.359,E2 19325.359} C_VEL
LIN {X 0,Y 409.389,Z 930.167,A -85,B 0,C 180,E1 19323.218,E2 19323.218} C_VEL
LIN {X 0,Y 411.972,Z 914.147,A -85,B 0,C 180,E1 19321.28,E2 19321.28} C_VEL
LIN {X 0,Y 414.704,Z 896.485,A -85,B 0,C 180,E1 19319.502,E2 19319.502} C_VEL
LIN {X 0,Y 417.404,Z 877.724,A -85,B 0,C 180,E1 19317.956,E2 19317.956} C_VEL
LIN {X 0,Y 419.826,Z 859.084,A -85,B 0,C 180,E1 19316.714,E2 19316.714} C_VEL
LIN {X 0,Y 422.019,Z 839.442,A -85,B 0,C 180,E1 19315.677,E2 19315.677} C_VEL
LIN {X 0,Y 423.917,Z 818.715,A -85,B 0,C 180,E1 19314.858,E2 19314.858} C_VEL
LIN {X 0,Y 425.277,Z 797.995,A -85,B 0,C 180,E1 19314.293,E2 19314.293} C_VEL
LIN {X 0,Y 426.452,Z 768.552,A -85,B 0,C 180,E1 19313.774,E2 19313.774} C_VEL
LIN {X 0,Y 428.929,Z 746.073,A -85,B 0,C 180,E1 19313.53,E2 19313.53} C_VEL
LIN {X 0,Y 442.589,Z 715.678,A -85,B 0,C 180,E1 19311.923,E2 19311.923} C_VEL
LIN {X 0,Y 452.611,Z 697.5,A -85,B 0,C 180,E1 19311.144,E2 19311.144} C_VEL
LIN {X 0,Y 456.754,Z 690.762,A -85,B 0,C 180,E1 19310.898,E2 19310.898} C_VEL
LIN {X 0,Y 447.758,Z 677,A -85,B 0,C 180,E1 19309.005,E2 19309.005} C_VEL
LIN {X 0,Y 441.287,Z 663.152,A -85,B 0,C 180,E1 19307.232,E2 19307.232} C_VEL
LIN {X 0,Y 436.618,Z 647.885,A -85,B 0,C 180,E1 19305.413,E2 19305.413} C_VEL
LIN {X 0,Y 433.662,Z 630.438,A -85,B 0,C 180,E1 19303.481,E2 19303.481} C_VEL
LIN {X 0,Y 432.754,Z 612.28,A -85,B 0,C 180,E1 19301.625,E2 19301.625} C_VEL
LIN {X 0,Y 433.967,Z 589.458,A -85,B 0,C 180,E1 19299.482,E2 19299.482} C_VEL
LIN {X 0,Y 439.555,Z 545.709,A -85,B 0,C 180,E1 19295.614,E2 19295.614} C_VEL
LIN {X 0,Y 439.77,Z 543.752,A -85,B 0,C 180,E1 19295.434,E2 19295.434} C_VEL
LIN {X 0,Y 430.059,Z 522.878,A -85,B 0,C 180,E1 19291.854,E2 19291.854} C_VEL
LIN {X 0,Y 421.049,Z 504.382,A -85,B 0,C 180,E1 19288.355,E2 19288.355} C_VEL
LIN {X 0,Y 412.733,Z 487.803,A -85,B 0,C 180,E1 19284.93,E2 19284.93} C_VEL
LIN {X 0,Y 407.732,Z 478.26,A -85,B 0,C 180,E1 19282.796,E2 19282.796} C_VEL
LIN {X 0,Y 405.606,Z 474.132,A -85,B 0,C 180,E1 19281.853,E2 19281.853} C_VEL
LIN {X 0,Y 403.602,Z 469.997,A -85,B 0,C 180,E1 19280.9,E2 19280.9} C_VEL
LIN {X 0,Y 401.735,Z 466.755,A -85,B 0,C 180,E1 19280.088,E2 19280.088} C_VEL
LIN {X 0,Y 401.482,Z 465.474,A -85,B 0,C 180,E1 19279.797,E2 19279.797} C_VEL
LIN {X 0,Y 401.503,Z 465.476,A -85,B 0,C 180,E1 19275.898,E2 19275.898} C_VEL
LIN {X 0,Y 401.457,Z 465.482,A -85,B 0,C 180,E1 19272.076,E2 19272.076} C_VEL
LIN {X 0,Y 401.499,Z 465.478,A -85,B 0,C 180,E1 19268.16,E2 19268.16} C_VEL
LIN {X 0,Y 401.463,Z 465.48,A -85,B 0,C 180,E1 19264.285,E2 19264.285} C_VEL
LIN {X 0,Y 401.489,Z 465.472,A -85,B 0,C 180,E1 19260.142,E2 19260.142} C_VEL
LIN {X 0,Y 401.478,Z 465.473,A -85,B 0,C 180,E1 19256.287,E2 19256.287} C_VEL
LIN {X 0,Y 401.481,Z 465.453,A -85,B 0,C 180,E1 19252.271,E2 19252.271} C_VEL
LIN {X 0,Y 401.501,Z 465.465,A -85,B 0,C 180,E1 19248.363,E2 19248.363} C_VEL
LIN {X 0,Y 401.491,Z 465.474,A -85,B 0,C 180,E1 19244.249,E2 19244.249} C_VEL
LIN {X 0,Y 401.504,Z 465.469,A -85,B 0,C 180,E1 19240.274,E2 19240.274} C_VEL
LIN {X 0,Y 401.5,Z 465.464,A -85,B 0,C 180,E1 19236.207,E2 19236.207} C_VEL
LIN {X 0,Y 401.495,Z 465.463,A -85,B 0,C 180,E1 19232.245,E2 19232.245} C_VEL
LIN {X 0,Y 401.492,Z 465.465,A -85,B 0,C 180,E1 19228.3,E2 19228.3} C_VEL
LIN {X 0,Y 401.489,Z 465.469,A -85,B 0,C 180,E1 19224.522,E2 19224.522} C_VEL
LIN {X 0,Y 401.459,Z 465.48,A -85,B 0,C 180,E1 19220.539,E2 19220.539} C_VEL
LIN {X 0,Y 401.503,Z 465.575,A -85,B 0,C 180,E1 19218.515,E2 19218.515} C_VEL
LIN {X 0,Y 402.882,Z 469.059,A -85,B 0,C 180,E1 19217.905,E2 19217.905} C_VEL
LIN {X 0,Y 404.017,Z 471.118,A -85,B 0,C 180,E1 19217.497,E2 19217.497} C_VEL
LIN {X 0,Y 410.008,Z 483.319,A -85,B 0,C 180,E1 19215.288,E2 19215.288} C_VEL
LIN {X 0,Y 417.622,Z 499.996,A -85,B 0,C 180,E1 19212.59,E2 19212.59} C_VEL
LIN {X 0,Y 418.97,Z 502.681,A -85,B 0,C 180,E1 19212.259,E2 19212.259} C_VEL
LIN {X 0,Y 430.436,Z 522.597,A -85,B 0,C 180,E1 19210.444,E2 19210.444} C_VEL
LIN {X 0,Y 432.681,Z 527.213,A -85,B 0,C 180,E1 19210.09,E2 19210.09} C_VEL
LIN {X 0,Y 433.421,Z 533.102,A -85,B 0,C 180,E1 19209.881,E2 19209.881} C_VEL
LIN {X 0,Y 426.717,Z 762.108,A -85,B 0,C 180,E1 19205.764,E2 19205.764} C_VEL
LIN {X 0,Y 425.512,Z 782.695,A -85,B 0,C 180,E1 19205.171,E2 19205.171} C_VEL
LIN {X 0,Y 423.776,Z 803.26,A -85,B 0,C 180,E1 19204.325,E2 19204.325} C_VEL
LIN {X 0,Y 421.69,Z 822.91,A -85,B 0,C 180,E1 19203.251,E2 19203.251} C_VEL
LIN {X 0,Y 419.392,Z 840.954,A -85,B 0,C 180,E1 19202.015,E2 19202.015} C_VEL
LIN {X 0,Y 416.755,Z 859.036,A -85,B 0,C 180,E1 19200.491,E2 19200.491} C_VEL
LIN {X 0,Y 416.078,Z 863.292,A -85,B 0,C 180,E1 19200.078,E2 19200.078} C_VEL
LIN {X 0,Y 414.202,Z 869.687,A -85,B 0,C 180,E1 19199.512,E2 19199.512} C_VEL
LIN {X 0,Y 406.224,Z 885.403,A -85,B 0,C 180,E1 19198.151,E2 19198.151} C_VEL
LIN {X 0,Y 404.311,Z 891.105,A -85,B 0,C 180,E1 19197.475,E2 19197.475} C_VEL
LIN {X 0,Y 401.459,Z 906.491,A -85,B 0,C 180,E1 19195.206,E2 19195.206} C_VEL
LIN {X 0,Y 399.003,Z 919.808,A -85,B 0,C 180,E1 19192.855,E2 19192.855} C_VEL
LIN {X 0,Y 396.883,Z 931.726,A -85,B 0,C 180,E1 19190.343,E2 19190.343} C_VEL
LIN {X 0,Y 395.145,Z 942.235,A -85,B 0,C 180,E1 19187.676,E2 19187.676} C_VEL
LIN {X 0,Y 393.764,Z 951.69,A -85,B 0,C 180,E1 19184.709,E2 19184.709} C_VEL
LIN {X 0,Y 392.865,Z 959.117,A -85,B 0,C 180,E1 19181.747,E2 19181.747} C_VEL
LIN {X 0,Y 392.366,Z 964.723,A -85,B 0,C 180,E1 19178.794,E2 19178.794} C_VEL
LIN {X 0,Y 392.112,Z 968.656,A -85,B 0,C 180,E1 19175.853,E2 19175.853} C_VEL
LIN {X 0,Y 392.021,Z 971.016,A -85,B 0,C 180,E1 19172.923,E2 19172.923} C_VEL
LIN {X 0,Y 392.012,Z 971.842,A -85,B 0,C 180,E1 19169.999,E2 19169.999} C_VEL
LIN {X 0,Y 392.018,Z 971.057,A -85,B 0,C 180,E1 19167.075,E2 19167.075} C_VEL
LIN {X 0,Y 392.106,Z 968.753,A -85,B 0,C 180,E1 19164.145,E2 19164.145} C_VEL
LIN {X 0,Y 392.357,Z 964.873,A -85,B 0,C 180,E1 19161.204,E2 19161.204} C_VEL
LIN {X 0,Y 392.845,Z 959.321,A -85,B 0,C 180,E1 19158.251,E2 19158.251} C_VEL
LIN {X 0,Y 393.733,Z 951.953,A -85,B 0,C 180,E1 19155.288,E2 19155.288} C_VEL
LIN {X 0,Y 395.099,Z 942.549,A -85,B 0,C 180,E1 19152.321,E2 19152.321} C_VEL
LIN {X 0,Y 396.867,Z 931.832,A -85,B 0,C 180,E1 19149.589,E2 19149.589} C_VEL
LIN {X 0,Y 398.924,Z 920.252,A -85,B 0,C 180,E1 19147.139,E2 19147.139} C_VEL
LIN {X 0,Y 401.478,Z 906.454,A -85,B 0,C 180,E1 19144.694,E2 19144.694} C_VEL
LIN {X 0,Y 404.292,Z 891.27,A -85,B 0,C 180,E1 19142.452,E2 19142.452} C_VEL
LIN {X 0,Y 407.14,Z 875.449,A -85,B 0,C 180,E1 19140.501,E2 19140.501} C_VEL
LIN {X 0,Y 409.948,Z 858.738,A -85,B 0,C 180,E1 19138.778,E2 19138.778} C_VEL
LIN {X 0,Y 412.781,Z 840.269,A -85,B 0,C 180,E1 19137.214,E2 19137.214} C_VEL
LIN {X 0,Y 415.292,Z 821.255,A -85,B 0,C 180,E1 19135.916,E2 19135.916} C_VEL
LIN {X 0,Y 417.412,Z 801.687,A -85,B 0,C 180,E1 19134.865,E2 19134.865} C_VEL
LIN {X 0,Y 419.113,Z 781.886,A -85,B 0,C 180,E1 19134.064,E2 19134.064} C_VEL
LIN {X 0,Y 420.353,Z 760.639,A -85,B 0,C 180,E1 19133.463,E2 19133.463} C_VEL
LIN {X 0,Y 426.888,Z 544.535,A -85,B 0,C 180,E1 19129.525,E2 19129.525} C_VEL
LIN {X 0,Y 422.836,Z 529.109,A -85,B 0,C 180,E1 19128.709,E2 19128.709} C_VEL
LIN {X 0,Y 411.083,Z 508.463,A -85,B 0,C 180,E1 19126.758,E2 19126.758} C_VEL
LIN {X 0,Y 408.304,Z 503.802,A -85,B 0,C 180,E1 19126.253,E2 19126.253} C_VEL
LIN {X 0,Y 403.095,Z 489.599,A -85,B 0,C 180,E1 19123.382,E2 19123.382} C_VEL
LIN {X 0,Y 398.55,Z 478.298,A -85,B 0,C 180,E1 19120.808,E2 19120.808} C_VEL
LIN {X 0,Y 398.213,Z 478.201,A -85,B 0,C 180,E1 19120.686,E2 19120.686} C_VEL
LIN {X 0,Y 404.756,Z 494.903,A -85,B 0,C 180,E1 19117.601,E2 19117.601} C_VEL
LIN {X 0,Y 411.22,Z 513.135,A -85,B 0,C 180,E1 19114.485,E2 19114.485} C_VEL
LIN {X 0,Y 414.155,Z 522.564,A -85,B 0,C 180,E1 19112.984,E2 19112.984} C_VEL
LIN {X 0,Y 410.822,Z 557.765,A -85,B 0,C 180,E1 19108.969,E2 19108.969} C_VEL
LIN {X 0,Y 407.842,Z 592.956,A -85,B 0,C 180,E1 19105.018,E2 19105.018} C_VEL
LIN {X 0,Y 405.524,Z 624.229,A -85,B 0,C 180,E1 19101.6,E2 19101.6} C_VEL
LIN {X 0,Y 406.147,Z 630.851,A -85,B 0,C 180,E1 19101.378,E2 19101.378} C_VEL
LIN {X 0,Y 401.17,Z 764.248,A -85,B 0,C 180,E1 19098.007,E2 19098.007} C_VEL
LIN {X 0,Y 400.752,Z 780.82,A -85,B 0,C 180,E1 19097.384,E2 19097.384} C_VEL
LIN {X 0,Y 400.047,Z 797.323,A -85,B 0,C 180,E1 19096.48,E2 19096.48} C_VEL
LIN {X 0,Y 399.221,Z 812.175,A -85,B 0,C 180,E1 19095.396,E2 19095.396} C_VEL
LIN {X 0,Y 398.176,Z 827.555,A -85,B 0,C 180,E1 19093.95,E2 19093.95} C_VEL
LIN {X 0,Y 397.131,Z 841.002,A -85,B 0,C 180,E1 19092.344,E2 19092.344} C_VEL
LIN {X 0,Y 396.194,Z 852.708,A -85,B 0,C 180,E1 19090.616,E2 19090.616} C_VEL
LIN {X 0,Y 395.3,Z 863.686,A -85,B 0,C 180,E1 19088.583,E2 19088.583} C_VEL
LIN {X 0,Y 394.643,Z 872.453,A -85,B 0,C 180,E1 19086.547,E2 19086.547} C_VEL
LIN {X 0,Y 394.127,Z 880.162,A -85,B 0,C 180,E1 19084.219,E2 19084.219} C_VEL
LIN {X 0,Y 393.846,Z 885.514,A -85,B 0,C 180,E1 19082.037,E2 19082.037} C_VEL
LIN {X 0,Y 393.739,Z 889.595,A -85,B 0,C 180,E1 19079.564,E2 19079.564} C_VEL
LIN {X 0,Y 393.803,Z 891.647,A -85,B 0,C 180,E1 19077.235,E2 19077.235} C_VEL
LIN {X 0,Y 394.047,Z 892,A -85,B 0,C 180,E1 19074.759,E2 19074.759} C_VEL
LIN {X 0,Y 394.49,Z 890.416,A -85,B 0,C 180,E1 19072.319,E2 19072.319} C_VEL
LIN {X 0,Y 395.16,Z 887.096,A -85,B 0,C 180,E1 19069.946,E2 19069.946} C_VEL
LIN {X 0,Y 396.112,Z 881.919,A -85,B 0,C 180,E1 19067.611,E2 19067.611} C_VEL
LIN {X 0,Y 397.172,Z 875.646,A -85,B 0,C 180,E1 19065.568,E2 19065.568} C_VEL
LIN {X 0,Y 398.626,Z 866.819,A -85,B 0,C 180,E1 19063.369,E2 19063.369} C_VEL
LIN {X 0,Y 400.11,Z 857.084,A -85,B 0,C 180,E1 19061.496,E2 19061.496} C_VEL
LIN {X 0,Y 401.693,Z 845.76,A -85,B 0,C 180,E1 19059.758,E2 19059.758} C_VEL
LIN {X 0,Y 403.289,Z 832.747,A -85,B 0,C 180,E1 19058.168,E2 19058.168} C_VEL
LIN {X 0,Y 404.737,Z 818.126,A -85,B 0,C 180,E1 19056.78,E2 19056.78} C_VEL
LIN {X 0,Y 405.846,Z 803.4,A -85,B 0,C 180,E1 19055.706,E2 19055.706} C_VEL
LIN {X 0,Y 406.625,Z 788.12,A -85,B 0,C 180,E1 19054.878,E2 19054.878} C_VEL
LIN {X 0,Y 408.561,Z 757.794,A -85,B 0,C 180,E1 19053.613,E2 19053.613} C_VEL
LIN {X 0,Y 420.371,Z 663.416,A -85,B 0,C 180,E1 19050.034,E2 19050.034} C_VEL
LIN {X 0,Y 428.447,Z 648.721,A -85,B 0,C 180,E1 19048.797,E2 19048.797} C_VEL
LIN {X 0,Y 436.551,Z 628.984,A -85,B 0,C 180,E1 19045.707,E2 19045.707} C_VEL
LIN {X 0,Y 445.434,Z 613.385,A -85,B 0,C 180,E1 19043.046,E2 19043.046} C_VEL
LIN {X 0,Y 448.213,Z 609.44,A -85,B 0,C 180,E1 19042.303,E2 19042.303} C_VEL
LIN {X 0,Y 440.67,Z 620.781,A -85,B 0,C 180,E1 19040.485,E2 19040.485} C_VEL
LIN {X 0,Y 435.448,Z 632.155,A -85,B 0,C 180,E1 19038.602,E2 19038.602} C_VEL
LIN {X 0,Y 432.637,Z 643.645,A -85,B 0,C 180,E1 19036.655,E2 19036.655} C_VEL
LIN {X 0,Y 432.205,Z 655.169,A -85,B 0,C 180,E1 19034.691,E2 19034.691} C_VEL
LIN {X 0,Y 434.17,Z 666.756,A -85,B 0,C 180,E1 19032.724,E2 19032.724} C_VEL
LIN {X 0,Y 438.514,Z 678.15,A -85,B 0,C 180,E1 19030.8,E2 19030.8} C_VEL
LIN {X 0,Y 445.32,Z 689.488,A -85,B 0,C 180,E1 19028.916,E2 19028.916} C_VEL
LIN {X 0,Y 434.75,Z 708.679,A -85,B 0,C 180,E1 19028.136,E2 19028.136} C_VEL
LIN {X 0,Y 426.859,Z 725.875,A -85,B 0,C 180,E1 19027.266,E2 19027.266} C_VEL
LIN {X 0,Y 425.567,Z 729.277,A -85,B 0,C 180,E1 19027.125,E2 19027.125} C_VEL
LIN {X 0,Y 422.19,Z 750.214,A -85,B 0,C 180,E1 19027.034,E2 19027.034} C_VEL
LIN {X 0,Y 419.783,Z 773.268,A -85,B 0,C 180,E1 19026.799,E2 19026.799} C_VEL
LIN {X 0,Y 418.6,Z 802.721,A -85,B 0,C 180,E1 19026.229,E2 19026.229} C_VEL
LIN {X 0,Y 417.016,Z 823.553,A -85,B 0,C 180,E1 19025.6,E2 19025.6} C_VEL
LIN {X 0,Y 414.939,Z 844.02,A -85,B 0,C 180,E1 19024.718,E2 19024.718} C_VEL
LIN {X 0,Y 412.505,Z 863.629,A -85,B 0,C 180,E1 19023.599,E2 19023.599} C_VEL
LIN {X 0,Y 409.924,Z 881.901,A -85,B 0,C 180,E1 19022.288,E2 19022.288} C_VEL
LIN {X 0,Y 406.99,Z 900.556,A -85,B 0,C 180,E1 19020.649,E2 19020.649} C_VEL
LIN {X 0,Y 404.106,Z 918.113,A -85,B 0,C 180,E1 19018.767,E2 19018.767} C_VEL
LIN {X 0,Y 401.366,Z 934.049,A -85,B 0,C 180,E1 19016.722,E2 19016.722} C_VEL
LIN {X 0,Y 398.985,Z 948.371,A -85,B 0,C 180,E1 19014.539,E2 19014.539} C_VEL
LIN {X 0,Y 396.751,Z 962.064,A -85,B 0,C 180,E1 19012.056,E2 19012.056} C_VEL
LIN {X 0,Y 394.95,Z 974.374,A -85,B 0,C 180,E1 19009.369,E2 19009.369} C_VEL
LIN {X 0,Y 393.695,Z 984.576,A -85,B 0,C 180,E1 19006.678,E2 19006.678} C_VEL
LIN {X 0,Y 392.802,Z 993.374,A -85,B 0,C 180,E1 19003.844,E2 19003.844} C_VEL
LIN {X 0,Y 392.323,Z 1000.676,A -85,B 0,C 180,E1 19000.871,E2 19000.871} C_VEL
LIN {X 0,Y 392.158,Z 1005.918,A -85,B 0,C 180,E1 18998.062,E2 18998.062} C_VEL
LIN {X 0,Y 392.115,Z 1009.519,A -85,B 0,C 180,E1 18995.268,E2 18995.268} C_VEL
LIN {X 0,Y 392.162,Z 1011.577,A -85,B 0,C 180,E1 18992.485,E2 18992.485} C_VEL
LIN {X 0,Y 392.183,Z 1012.192,A -85,B 0,C 180,E1 18989.709,E2 18989.709} C_VEL
LIN {X 0,Y 392.149,Z 1011.294,A -85,B 0,C 180,E1 18986.931,E2 18986.931} C_VEL
LIN {X 0,Y 392.112,Z 1008.86,A -85,B 0,C 180,E1 18984.147,E2 18984.147} C_VEL
LIN {X 0,Y 392.155,Z 1004.675,A -85,B 0,C 180,E1 18981.201,E2 18981.201} C_VEL
LIN {X 0,Y 392.394,Z 999.081,A -85,B 0,C 180,E1 18978.388,E2 18978.388} C_VEL
LIN {X 0,Y 392.967,Z 991.298,A -85,B 0,C 180,E1 18975.411,E2 18975.411} C_VEL
LIN {X 0,Y 393.943,Z 981.941,A -85,B 0,C 180,E1 18972.574,E2 18972.574} C_VEL
LIN {X 0,Y 395.373,Z 971.131,A -85,B 0,C 180,E1 18969.884,E2 18969.884} C_VEL
LIN {X 0,Y 397.187,Z 958.924,A -85,B 0,C 180,E1 18967.347,E2 18967.347} C_VEL
LIN {X 0,Y 399.415,Z 945.334,A -85,B 0,C 180,E1 18964.973,E2 18964.973} C_VEL
LIN {X 0,Y 401.972,Z 930.313,A -85,B 0,C 180,E1 18962.763,E2 18962.763} C_VEL
LIN {X 0,Y 404.792,Z 913.735,A -85,B 0,C 180,E1 18960.721,E2 18960.721} C_VEL
LIN {X 0,Y 407.686,Z 896.078,A -85,B 0,C 180,E1 18958.919,E2 18958.919} C_VEL
LIN {X 0,Y 410.528,Z 877.322,A -85,B 0,C 180,E1 18957.353,E2 18957.353} C_VEL
LIN {X 0,Y 413.073,Z 858.688,A -85,B 0,C 180,E1 18956.096,E2 18956.096} C_VEL
LIN {X 0,Y 415.372,Z 839.063,A -85,B 0,C 180,E1 18955.048,E2 18955.048} C_VEL
LIN {X 0,Y 417.384,Z 818.152,A -85,B 0,C 180,E1 18954.216,E2 18954.216} C_VEL
LIN {X 0,Y 418.796,Z 797.367,A -85,B 0,C 180,E1 18953.645,E2 18953.645} C_VEL
LIN {X 0,Y 420.006,Z 768.526,A -85,B 0,C 180,E1 18953.132,E2 18953.132} C_VEL
LIN {X 0,Y 422.835,Z 743.464,A -85,B 0,C 180,E1 18952.874,E2 18952.874} C_VEL
LIN {X 0,Y 436.506,Z 713.649,A -85,B 0,C 180,E1 18951.294,E2 18951.294} C_VEL
LIN {X 0,Y 446.583,Z 695.602,A -85,B 0,C 180,E1 18950.518,E2 18950.518} C_VEL
LIN {X 0,Y 448.309,Z 692.72,A -85,B 0,C 180,E1 18950.406,E2 18950.406} C_VEL
LIN {X 0,Y 439.822,Z 678.874,A -85,B 0,C 180,E1 18948.509,E2 18948.509} C_VEL
LIN {X 0,Y 433.628,Z 664.516,A -85,B 0,C 180,E1 18946.675,E2 18946.675} C_VEL
LIN {X 0,Y 429.079,Z 647.967,A -85,B 0,C 180,E1 18944.707,E2 18944.707} C_VEL
LIN {X 0,Y 426.536,Z 630.113,A -85,B 0,C 180,E1 18942.736,E2 18942.736} C_VEL
LIN {X 0,Y 426.072,Z 610.225,A -85,B 0,C 180,E1 18940.715,E2 18940.715} C_VEL
LIN {X 0,Y 427.942,Z 586.497,A -85,B 0,C 180,E1 18938.492,E2 18938.492} C_VEL
LIN {X 0,Y 433.214,Z 547.833,A -85,B 0,C 180,E1 18935.037,E2 18935.037} C_VEL
LIN {X 0,Y 425.045,Z 529.871,A -85,B 0,C 180,E1 18931.957,E2 18931.957} C_VEL
LIN {X 0,Y 415.699,Z 510.44,A -85,B 0,C 180,E1 18928.283,E2 18928.283} C_VEL
LIN {X 0,Y 407.041,Z 493.168,A -85,B 0,C 180,E1 18924.682,E2 18924.682} C_VEL
LIN {X 0,Y 400.262,Z 479.984,A -85,B 0,C 180,E1 18921.697,E2 18921.697} C_VEL
LIN {X 0,Y 397.855,Z 475.398,A -85,B 0,C 180,E1 18920.6,E2 18920.6} C_VEL
LIN {X 0,Y 396.089,Z 471.976,A -85,B 0,C 180,E1 18919.771,E2 18919.771} C_VEL
LIN {X 0,Y 393.739,Z 467.562,A -85,B 0,C 180,E1 18918.66,E2 18918.66} C_VEL
LIN {X 0,Y 393.531,Z 466.465,A -85,B 0,C 180,E1 18918.414,E2 18918.414} C_VEL
LIN {X 0,Y 393.556,Z 466.463,A -85,B 0,C 180,E1 18914.546,E2 18914.546} C_VEL
LIN {X 0,Y 393.52,Z 466.47,A -85,B 0,C 180,E1 18910.393,E2 18910.393} C_VEL
LIN {X 0,Y 393.562,Z 466.464,A -85,B 0,C 180,E1 18906.418,E2 18906.418} C_VEL
LIN {X 0,Y 393.518,Z 466.468,A -85,B 0,C 180,E1 18902.33,E2 18902.33} C_VEL
LIN {X 0,Y 393.562,Z 466.459,A -85,B 0,C 180,E1 18898.398,E2 18898.398} C_VEL
LIN {X 0,Y 393.529,Z 466.465,A -85,B 0,C 180,E1 18894.459,E2 18894.459} C_VEL
LIN {X 0,Y 393.563,Z 466.454,A -85,B 0,C 180,E1 18890.642,E2 18890.642} C_VEL
LIN {X 0,Y 393.546,Z 466.443,A -85,B 0,C 180,E1 18886.632,E2 18886.632} C_VEL
LIN {X 0,Y 393.564,Z 466.446,A -85,B 0,C 180,E1 18882.708,E2 18882.708} C_VEL
LIN {X 0,Y 393.526,Z 466.464,A -85,B 0,C 180,E1 18878.82,E2 18878.82} C_VEL
LIN {X 0,Y 393.559,Z 466.465,A -85,B 0,C 180,E1 18874.895,E2 18874.895} C_VEL
LIN {X 0,Y 393.524,Z 466.47,A -85,B 0,C 180,E1 18870.929,E2 18870.929} C_VEL
LIN {X 0,Y 393.549,Z 466.468,A -85,B 0,C 180,E1 18866.891,E2 18866.891} C_VEL
LIN {X 0,Y 393.536,Z 466.462,A -85,B 0,C 180,E1 18862.976,E2 18862.976} C_VEL
LIN {X 0,Y 393.598,Z 466.692,A -85,B 0,C 180,E1 18859.687,E2 18859.687} C_VEL
LIN {X 0,Y 395.035,Z 470.209,A -85,B 0,C 180,E1 18859.039,E2 18859.039} C_VEL
LIN {X 0,Y 396.052,Z 471.82,A -85,B 0,C 180,E1 18858.687,E2 18858.687} C_VEL
LIN {X 0,Y 402.737,Z 485.239,A -85,B 0,C 180,E1 18856.159,E2 18856.159} C_VEL
LIN {X 0,Y 410.412,Z 501.833,A -85,B 0,C 180,E1 18853.385,E2 18853.385} C_VEL
LIN {X 0,Y 422.136,Z 521.72,A -85,B 0,C 180,E1 18851.439,E2 18851.439} C_VEL
LIN {X 0,Y 426.928,Z 530.966,A -85,B 0,C 180,E1 18850.667,E2 18850.667} C_VEL
LIN {X 0,Y 427.261,Z 535.035,A -85,B 0,C 180,E1 18850.539,E2 18850.539} C_VEL
LIN {X 0,Y 420.247,Z 762.627,A -85,B 0,C 180,E1 18846.397,E2 18846.397} C_VEL
LIN {X 0,Y 418.985,Z 783.234,A -85,B 0,C 180,E1 18845.795,E2 18845.795} C_VEL
LIN {X 0,Y 417.185,Z 803.639,A -85,B 0,C 180,E1 18844.945,E2 18844.945} C_VEL
LIN {X 0,Y 415.074,Z 822.755,A -85,B 0,C 180,E1 18843.893,E2 18843.893} C_VEL
LIN {X 0,Y 412.67,Z 840.903,A -85,B 0,C 180,E1 18842.643,E2 18842.643} C_VEL
LIN {X 0,Y 409.827,Z 859.438,A -85,B 0,C 180,E1 18841.063,E2 18841.063} C_VEL
LIN {X 0,Y 406.924,Z 876.644,A -85,B 0,C 180,E1 18839.272,E2 18839.272} C_VEL
LIN {X 0,Y 404.311,Z 891.105,A -85,B 0,C 180,E1 18837.475,E2 18837.475} C_VEL
LIN {X 0,Y 402.394,Z 896.78,A -85,B 0,C 180,E1 18836.763,E2 18836.763} C_VEL
LIN {X 0,Y 394.317,Z 910.68,A -85,B 0,C 180,E1 18835.013,E2 18835.013} C_VEL
LIN {X 0,Y 392.433,Z 915.59,A -85,B 0,C 180,E1 18834.197,E2 18834.197} C_VEL
LIN {X 0,Y 390.007,Z 928.143,A -85,B 0,C 180,E1 18831.664,E2 18831.664} C_VEL
LIN {X 0,Y 387.969,Z 939.323,A -85,B 0,C 180,E1 18828.947,E2 18828.947} C_VEL
LIN {X 0,Y 386.452,Z 948.556,A -85,B 0,C 180,E1 18826.225,E2 18826.225} C_VEL
LIN {X 0,Y 385.333,Z 956.495,A -85,B 0,C 180,E1 18823.332,E2 18823.332} C_VEL
LIN {X 0,Y 384.616,Z 962.846,A -85,B 0,C 180,E1 18820.333,E2 18820.333} C_VEL
LIN {X 0,Y 384.228,Z 967.505,A -85,B 0,C 180,E1 18817.325,E2 18817.325} C_VEL
LIN {X 0,Y 384.07,Z 970.55,A -85,B 0,C 180,E1 18814.329,E2 18814.329} C_VEL
LIN {X 0,Y 384.013,Z 972.058,A -85,B 0,C 180,E1 18811.342,E2 18811.342} C_VEL
LIN {X 0,Y 384.012,Z 972.05,A -85,B 0,C 180,E1 18808.507,E2 18808.507} C_VEL
LIN {X 0,Y 384.07,Z 970.509,A -85,B 0,C 180,E1 18805.52,E2 18805.52} C_VEL
LIN {X 0,Y 384.235,Z 967.397,A -85,B 0,C 180,E1 18802.5,E2 18802.5} C_VEL
LIN {X 0,Y 384.627,Z 962.726,A -85,B 0,C 180,E1 18799.515,E2 18799.515} C_VEL
LIN {X 0,Y 385.359,Z 956.29,A -85,B 0,C 180,E1 18796.495,E2 18796.495} C_VEL
LIN {X 0,Y 386.562,Z 947.932,A -85,B 0,C 180,E1 18793.469,E2 18793.469} C_VEL
LIN {X 0,Y 388.223,Z 937.98,A -85,B 0,C 180,E1 18790.595,E2 18790.595} C_VEL
LIN {X 0,Y 390.199,Z 927.182,A -85,B 0,C 180,E1 18788.03,E2 18788.03} C_VEL
LIN {X 0,Y 392.694,Z 914.324,A -85,B 0,C 180,E1 18785.478,E2 18785.478} C_VEL
LIN {X 0,Y 395.523,Z 899.909,A -85,B 0,C 180,E1 18783.095,E2 18783.095} C_VEL
LIN {X 0,Y 398.48,Z 884.686,A -85,B 0,C 180,E1 18780.993,E2 18780.993} C_VEL
LIN {X 0,Y 401.447,Z 868.59,A -85,B 0,C 180,E1 18779.131,E2 18779.131} C_VEL
LIN {X 0,Y 404.378,Z 851.336,A -85,B 0,C 180,E1 18777.475,E2 18777.475} C_VEL
LIN {X 0,Y 407.18,Z 832.641,A -85,B 0,C 180,E1 18776.012,E2 18776.012} C_VEL
LIN {X 0,Y 409.623,Z 813.684,A -85,B 0,C 180,E1 18774.825,E2 18774.825} C_VEL
LIN {X 0,Y 411.693,Z 793.703,A -85,B 0,C 180,E1 18773.852,E2 18773.852} C_VEL
LIN {X 0,Y 413.316,Z 772.517,A -85,B 0,C 180,E1 18773.101,E2 18773.101} C_VEL
LIN {X 0,Y 414.394,Z 749.681,A -85,B 0,C 180,E1 18772.576,E2 18772.576} C_VEL
LIN {X 0,Y 420.75,Z 546.258,A -85,B 0,C 180,E1 18768.842,E2 18768.842} C_VEL
LIN {X 0,Y 417.288,Z 533.138,A -85,B 0,C 180,E1 18768.124,E2 18768.124} C_VEL
LIN {X 0,Y 405.743,Z 512.877,A -85,B 0,C 180,E1 18766.146,E2 18766.146} C_VEL
LIN {X 0,Y 400.523,Z 504.07,A -85,B 0,C 180,E1 18765.152,E2 18765.152} C_VEL
LIN {X 0,Y 395.059,Z 489.703,A -85,B 0,C 180,E1 18762.121,E2 18762.121} C_VEL
LIN {X 0,Y 392.877,Z 484.31,A -85,B 0,C 180,E1 18760.849,E2 18760.849} C_VEL
LIN {X 0,Y 392.256,Z 483.97,A -85,B 0,C 180,E1 18760.654,E2 18760.654} C_VEL
LIN {X 0,Y 398.743,Z 500.701,A -85,B 0,C 180,E1 18757.541,E2 18757.541} C_VEL
LIN {X 0,Y 405.072,Z 518.905,A -85,B 0,C 180,E1 18754.42,E2 18754.42} C_VEL
LIN {X 0,Y 407.063,Z 525.969,A -85,B 0,C 180,E1 18753.297,E2 18753.297} C_VEL
LIN {X 0,Y 403.622,Z 560.532,A -85,B 0,C 180,E1 18749.309,E2 18749.309} C_VEL
LIN {X 0,Y 400.477,Z 596.151,A -85,B 0,C 180,E1 18745.273,E2 18745.273} C_VEL
LIN {X 0,Y 398.248,Z 625.379,A -85,B 0,C 180,E1 18742.054,E2 18742.054} C_VEL
LIN {X 0,Y 398.839,Z 631.805,A -85,B 0,C 180,E1 18741.832,E2 18741.832} C_VEL
LIN {X 0,Y 393.569,Z 764.647,A -85,B 0,C 180,E1 18738.362,E2 18738.362} C_VEL
LIN {X 0,Y 393.139,Z 781.312,A -85,B 0,C 180,E1 18737.732,E2 18737.732} C_VEL
LIN {X 0,Y 392.403,Z 797.92,A -85,B 0,C 180,E1 18736.81,E2 18736.81} C_VEL
LIN {X 0,Y 391.53,Z 813.149,A -85,B 0,C 180,E1 18735.684,E2 18735.684} C_VEL
LIN {X 0,Y 390.454,Z 828.348,A -85,B 0,C 180,E1 18734.231,E2 18734.231} C_VEL
LIN {X 0,Y 389.404,Z 841.477,A -85,B 0,C 180,E1 18732.65,E2 18732.65} C_VEL
LIN {X 0,Y 388.386,Z 853.639,A -85,B 0,C 180,E1 18730.832,E2 18730.832} C_VEL
LIN {X 0,Y 387.512,Z 863.977,A -85,B 0,C 180,E1 18728.906,E2 18728.906} C_VEL
LIN {X 0,Y 386.767,Z 873.518,A -85,B 0,C 180,E1 18726.681,E2 18726.681} C_VEL
LIN {X 0,Y 386.227,Z 881.279,A -85,B 0,C 180,E1 18724.306,E2 18724.306} C_VEL
LIN {X 0,Y 385.939,Z 886.709,A -85,B 0,C 180,E1 18722.079,E2 18722.079} C_VEL
LIN {X 0,Y 385.833,Z 890.858,A -85,B 0,C 180,E1 18719.555,E2 18719.555} C_VEL
LIN {X 0,Y 385.915,Z 892.977,A -85,B 0,C 180,E1 18717.179,E2 18717.179} C_VEL
LIN {X 0,Y 386.187,Z 893.395,A -85,B 0,C 180,E1 18714.652,E2 18714.652} C_VEL
LIN {X 0,Y 386.652,Z 891.997,A -85,B 0,C 180,E1 18712.272,E2 18712.272} C_VEL
LIN {X 0,Y 387.366,Z 888.927,A -85,B 0,C 180,E1 18709.891,E2 18709.891} C_VEL
LIN {X 0,Y 388.374,Z 883.909,A -85,B 0,C 180,E1 18707.511,E2 18707.511} C_VEL
LIN {X 0,Y 389.609,Z 877.396,A -85,B 0,C 180,E1 18705.282,E2 18705.282} C_VEL
LIN {X 0,Y 391.165,Z 868.754,A -85,B 0,C 180,E1 18703.059,E2 18703.059} C_VEL
LIN {X 0,Y 392.917,Z 858.288,A -85,B 0,C 180,E1 18700.991,E2 18700.991} C_VEL
LIN {X 0,Y 394.56,Z 847.481,A -85,B 0,C 180,E1 18699.298,E2 18699.298} C_VEL
LIN {X 0,Y 396.277,Z 834.584,A -85,B 0,C 180,E1 18697.683,E2 18697.683} C_VEL
LIN {X 0,Y 397.845,Z 820.422,A -85,B 0,C 180,E1 18696.29,E2 18696.29} C_VEL
LIN {X 0,Y 399.165,Z 804.841,A -85,B 0,C 180,E1 18695.114,E2 18695.114} C_VEL
LIN {X 0,Y 400.067,Z 789.144,A -85,B 0,C 180,E1 18694.243,E2 18694.243} C_VEL
LIN {X 0,Y 402.373,Z 759.306,A -85,B 0,C 180,E1 18692.922,E2 18692.922} C_VEL
LIN {X 0,Y 414.182,Z 673.049,A -85,B 0,C 180,E1 18689.499,E2 18689.499} C_VEL
LIN {X 0,Y 415.172,Z 666.713,A -85,B 0,C 180,E1 18689.259,E2 18689.259} C_VEL
LIN {X 0,Y 423.723,Z 651.738,A -85,B 0,C 180,E1 18688.012,E2 18688.012} C_VEL
LIN {X 0,Y 431.861,Z 633.789,A -85,B 0,C 180,E1 18685.12,E2 18685.12} C_VEL
LIN {X 0,Y 440.87,Z 619.204,A -85,B 0,C 180,E1 18682.569,E2 18682.569} C_VEL
LIN {X 0,Y 441.629,Z 618.147,A -85,B 0,C 180,E1 18682.359,E2 18682.359} C_VEL
LIN {X 0,Y 433.814,Z 630.218,A -85,B 0,C 180,E1 18680.338,E2 18680.338} C_VEL
LIN {X 0,Y 429.144,Z 641.314,A -85,B 0,C 180,E1 18678.409,E2 18678.409} C_VEL
LIN {X 0,Y 426.785,Z 652.741,A -85,B 0,C 180,E1 18676.38,E2 18676.38} C_VEL
LIN {X 0,Y 426.858,Z 663.874,A -85,B 0,C 180,E1 18674.404,E2 18674.404} C_VEL
LIN {X 0,Y 429.289,Z 675.161,A -85,B 0,C 180,E1 18672.411,E2 18672.411} C_VEL
LIN {X 0,Y 433.956,Z 686.057,A -85,B 0,C 180,E1 18670.506,E2 18670.506} C_VEL
LIN {X 0,Y 437.333,Z 692.119,A -85,B 0,C 180,E1 18669.485,E2 18669.485} C_VEL
LIN {X 0,Y 427.148,Z 711.052,A -85,B 0,C 180,E1 18668.682,E2 18668.682} C_VEL
LIN {X 0,Y 419.206,Z 728.862,A -85,B 0,C 180,E1 18667.789,E2 18667.789} C_VEL
LIN {X 0,Y 415.816,Z 750.115,A -85,B 0,C 180,E1 18667.697,E2 18667.697} C_VEL
LIN {X 0,Y 413.386,Z 773.284,A -85,B 0,C 180,E1 18667.46,E2 18667.46} C_VEL
LIN {X 0,Y 412.153,Z 802.378,A -85,B 0,C 180,E1 18666.89,E2 18666.89} C_VEL
LIN {X 0,Y 410.509,Z 823.095,A -85,B 0,C 180,E1 18666.258,E2 18666.258} C_VEL
LIN {X 0,Y 408.359,Z 843.338,A -85,B 0,C 180,E1 18665.379,E2 18665.379} C_VEL
LIN {X 0,Y 405.878,Z 862.505,A -85,B 0,C 180,E1 18664.279,E2 18664.279} C_VEL
LIN {X 0,Y 403.199,Z 880.604,A -85,B 0,C 180,E1 18662.979,E2 18662.979} C_VEL
LIN {X 0,Y 400.11,Z 899.416,A -85,B 0,C 180,E1 18661.319,E2 18661.319} C_VEL
LIN {X 0,Y 397.144,Z 916.477,A -85,B 0,C 180,E1 18659.486,E2 18659.486} C_VEL
LIN {X 0,Y 394.264,Z 932.485,A -85,B 0,C 180,E1 18657.427,E2 18657.427} C_VEL
LIN {X 0,Y 391.54,Z 947.719,A -85,B 0,C 180,E1 18655.082,E2 18655.082} C_VEL
LIN {X 0,Y 389.118,Z 961.646,A -85,B 0,C 180,E1 18652.512,E2 18652.512} C_VEL
LIN {X 0,Y 387.202,Z 973.956,A -85,B 0,C 180,E1 18649.773,E2 18649.773} C_VEL
LIN {X 0,Y 385.818,Z 984.232,A -85,B 0,C 180,E1 18647.007,E2 18647.007} C_VEL
LIN {X 0,Y 384.866,Z 992.955,A -85,B 0,C 180,E1 18644.136,E2 18644.136} C_VEL
LIN {X 0,Y 384.349,Z 1000.259,A -85,B 0,C 180,E1 18641.1,E2 18641.1} C_VEL
LIN {X 0,Y 384.164,Z 1005.503,A -85,B 0,C 180,E1 18638.231,E2 18638.231} C_VEL
LIN {X 0,Y 384.118,Z 1009.106,A -85,B 0,C 180,E1 18635.378,E2 18635.378} C_VEL
LIN {X 0,Y 384.17,Z 1011.165,A -85,B 0,C 180,E1 18632.537,E2 18632.537} C_VEL
LIN {X 0,Y 384.193,Z 1011.781,A -85,B 0,C 180,E1 18629.703,E2 18629.703} C_VEL
LIN {X 0,Y 384.156,Z 1010.882,A -85,B 0,C 180,E1 18626.868,E2 18626.868} C_VEL
LIN {X 0,Y 384.116,Z 1008.446,A -85,B 0,C 180,E1 18624.024,E2 18624.024} C_VEL
LIN {X 0,Y 384.16,Z 1004.259,A -85,B 0,C 180,E1 18621.017,E2 18621.017} C_VEL
LIN {X 0,Y 384.426,Z 998.663,A -85,B 0,C 180,E1 18618.144,E2 18618.144} C_VEL
LIN {X 0,Y 385.055,Z 990.878,A -85,B 0,C 180,E1 18615.105,E2 18615.105} C_VEL
LIN {X 0,Y 386.106,Z 981.519,A -85,B 0,C 180,E1 18612.208,E2 18612.208} C_VEL
LIN {X 0,Y 387.663,Z 970.56,A -85,B 0,C 180,E1 18609.43,E2 18609.43} C_VEL
LIN {X 0,Y 389.592,Z 958.504,A -85,B 0,C 180,E1 18606.881,E2 18606.881} C_VEL
LIN {X 0,Y 391.956,Z 944.915,A -85,B 0,C 180,E1 18604.463,E2 18604.463} C_VEL
LIN {X 0,Y 394.678,Z 929.897,A -85,B 0,C 180,E1 18602.217,E2 18602.217} C_VEL
LIN {X 0,Y 397.659,Z 913.323,A -85,B 0,C 180,E1 18600.143,E2 18600.143} C_VEL
LIN {X 0,Y 400.746,Z 895.477,A -85,B 0,C 180,E1 18598.298,E2 18598.298} C_VEL
LIN {X 0,Y 403.766,Z 876.537,A -85,B 0,C 180,E1 18596.7,E2 18596.7} C_VEL
LIN {X 0,Y 406.385,Z 858.182,A -85,B 0,C 180,E1 18595.452,E2 18595.452} C_VEL
LIN {X 0,Y 408.778,Z 838.684,A -85,B 0,C 180,E1 18594.4,E2 18594.4} C_VEL
LIN {X 0,Y 410.892,Z 817.746,A -85,B 0,C 180,E1 18593.559,E2 18593.559} C_VEL
LIN {X 0,Y 412.357,Z 797.055,A -85,B 0,C 180,E1 18592.984,E2 18592.984} C_VEL
LIN {X 0,Y 413.605,Z 768.626,A -85,B 0,C 180,E1 18592.473,E2 18592.473} C_VEL
LIN {X 0,Y 416.565,Z 742.003,A -85,B 0,C 180,E1 18592.219,E2 18592.219} C_VEL
LIN {X 0,Y 417.186,Z 739.94,A -85,B 0,C 180,E1 18592.154,E2 18592.154} C_VEL
LIN {X 0,Y 430.688,Z 711.19,A -85,B 0,C 180,E1 18590.63,E2 18590.63} C_VEL
LIN {X 0,Y 439.893,Z 694.546,A -85,B 0,C 180,E1 18589.894,E2 18589.894} C_VEL
LIN {X 0,Y 431.689,Z 680.127,A -85,B 0,C 180,E1 18587.93,E2 18587.93} C_VEL
LIN {X 0,Y 425.809,Z 665.172,A -85,B 0,C 180,E1 18586.03,E2 18586.03} C_VEL
LIN {X 0,Y 421.643,Z 648.154,A -85,B 0,C 180,E1 18584.011,E2 18584.011} C_VEL
LIN {X 0,Y 419.484,Z 629.536,A -85,B 0,C 180,E1 18581.956,E2 18581.956} C_VEL
LIN {X 0,Y 419.506,Z 609.065,A -85,B 0,C 180,E1 18579.875,E2 18579.875} C_VEL
LIN {X 0,Y 421.936,Z 584.243,A -85,B 0,C 180,E1 18577.555,E2 18577.555} C_VEL
LIN {X 0,Y 426.642,Z 551.438,A -85,B 0,C 180,E1 18574.593,E2 18574.593} C_VEL
LIN {X 0,Y 417.646,Z 531.766,A -85,B 0,C 180,E1 18571.138,E2 18571.138} C_VEL
LIN {X 0,Y 408.376,Z 512.548,A -85,B 0,C 180,E1 18567.406,E2 18567.406} C_VEL
LIN {X 0,Y 400.674,Z 497.338,A -85,B 0,C 180,E1 18564.158,E2 18564.158} C_VEL
LIN {X 0,Y 394.569,Z 485.314,A -85,B 0,C 180,E1 18561.401,E2 18561.401} C_VEL
LIN {X 0,Y 391.788,Z 480.212,A -85,B 0,C 180,E1 18560.153,E2 18560.153} C_VEL
LIN {X 0,Y 389.775,Z 476.175,A -85,B 0,C 180,E1 18559.168,E2 18559.168} C_VEL
LIN {X 0,Y 387.48,Z 471.67,A -85,B 0,C 180,E1 18558.038,E2 18558.038} C_VEL
LIN {X 0,Y 385.779,Z 468.364,A -85,B 0,C 180,E1 18557.185,E2 18557.185} C_VEL
LIN {X 0,Y 385.609,Z 467.453,A -85,B 0,C 180,E1 18556.952,E2 18556.952} C_VEL
LIN {X 0,Y 385.613,Z 467.452,A -85,B 0,C 180,E1 18553.037,E2 18553.037} C_VEL
LIN {X 0,Y 385.609,Z 467.453,A -85,B 0,C 180,E1 18548.8,E2 18548.8} C_VEL
LIN {X 0,Y 385.619,Z 467.45,A -85,B 0,C 180,E1 18544.908,E2 18544.908} C_VEL
LIN {X 0,Y 385.612,Z 467.448,A -85,B 0,C 180,E1 18540.743,E2 18540.743} C_VEL
LIN {X 0,Y 385.62,Z 467.451,A -85,B 0,C 180,E1 18536.724,E2 18536.724} C_VEL
LIN {X 0,Y 385.615,Z 467.429,A -85,B 0,C 180,E1 18532.551,E2 18532.551} C_VEL
LIN {X 0,Y 385.623,Z 467.444,A -85,B 0,C 180,E1 18528.483,E2 18528.483} C_VEL
LIN {X 0,Y 385.619,Z 467.452,A -85,B 0,C 180,E1 18524.356,E2 18524.356} C_VEL
LIN {X 0,Y 385.627,Z 467.447,A -85,B 0,C 180,E1 18520.25,E2 18520.25} C_VEL
LIN {X 0,Y 385.619,Z 467.441,A -85,B 0,C 180,E1 18516.141,E2 18516.141} C_VEL
LIN {X 0,Y 385.624,Z 467.44,A -85,B 0,C 180,E1 18512.146,E2 18512.146} C_VEL
LIN {X 0,Y 385.624,Z 467.443,A -85,B 0,C 180,E1 18508.066,E2 18508.066} C_VEL
LIN {X 0,Y 385.617,Z 467.452,A -85,B 0,C 180,E1 18503.995,E2 18503.995} C_VEL
LIN {X 0,Y 385.59,Z 467.528,A -85,B 0,C 180,E1 18500.989,E2 18500.989} C_VEL
LIN {X 0,Y 386.937,Z 471.001,A -85,B 0,C 180,E1 18500.338,E2 18500.338} C_VEL
LIN {X 0,Y 388.2,Z 472.827,A -85,B 0,C 180,E1 18499.902,E2 18499.902} C_VEL
LIN {X 0,Y 395.122,Z 486.461,A -85,B 0,C 180,E1 18497.209,E2 18497.209} C_VEL
LIN {X 0,Y 401.998,Z 501.022,A -85,B 0,C 180,E1 18494.655,E2 18494.655} C_VEL
LIN {X 0,Y 403.473,Z 503.726,A -85,B 0,C 180,E1 18494.285,E2 18494.285} C_VEL
LIN {X 0,Y 414.745,Z 522.565,A -85,B 0,C 180,E1 18492.336,E2 18492.336} C_VEL
LIN {X 0,Y 421.229,Z 534.791,A -85,B 0,C 180,E1 18491.256,E2 18491.256} C_VEL
LIN {X 0,Y 413.838,Z 762.948,A -85,B 0,C 180,E1 18487.054,E2 18487.054} C_VEL
LIN {X 0,Y 412.525,Z 783.584,A -85,B 0,C 180,E1 18486.445,E2 18486.445} C_VEL
LIN {X 0,Y 410.646,Z 804.019,A -85,B 0,C 180,E1 18485.585,E2 18485.585} C_VEL
LIN {X 0,Y 408.439,Z 823.146,A -85,B 0,C 180,E1 18484.52,E2 18484.52} C_VEL
LIN {X 0,Y 405.888,Z 841.53,A -85,B 0,C 180,E1 18483.236,E2 18483.236} C_VEL
LIN {X 0,Y 402.973,Z 859.645,A -85,B 0,C 180,E1 18481.673,E2 18481.673} C_VEL
LIN {X 0,Y 400.014,Z 876.4,A -85,B 0,C 180,E1 18479.911,E2 18479.911} C_VEL
LIN {X 0,Y 397.028,Z 892.127,A -85,B 0,C 180,E1 18477.931,E2 18477.931} C_VEL
LIN {X 0,Y 394.14,Z 906.904,A -85,B 0,C 180,E1 18475.708,E2 18475.708} C_VEL
LIN {X 0,Y 392.433,Z 915.59,A -85,B 0,C 180,E1 18474.197,E2 18474.197} C_VEL
LIN {X 0,Y 390.575,Z 920.446,A -85,B 0,C 180,E1 18473.348,E2 18473.348} C_VEL
LIN {X 0,Y 382.681,Z 932.195,A -85,B 0,C 180,E1 18471.218,E2 18471.218} C_VEL
LIN {X 0,Y 380.959,Z 936.26,A -85,B 0,C 180,E1 18470.269,E2 18470.269} C_VEL
LIN {X 0,Y 379.155,Z 946.073,A -85,B 0,C 180,E1 18467.494,E2 18467.494} C_VEL
LIN {X 0,Y 377.741,Z 954.908,A -85,B 0,C 180,E1 18464.406,E2 18464.406} C_VEL
LIN {X 0,Y 376.839,Z 961.799,A -85,B 0,C 180,E1 18461.322,E2 18461.322} C_VEL
LIN {X 0,Y 376.349,Z 966.926,A -85,B 0,C 180,E1 18458.247,E2 18458.247} C_VEL
LIN {X 0,Y 376.114,Z 970.404,A -85,B 0,C 180,E1 18455.185,E2 18455.185} C_VEL
LIN {X 0,Y 376.039,Z 972.232,A -85,B 0,C 180,E1 18452.133,E2 18452.133} C_VEL
LIN {X 0,Y 376.027,Z 972.547,A -85,B 0,C 180,E1 18449.085,E2 18449.085} C_VEL
LIN {X 0,Y 376.068,Z 971.358,A -85,B 0,C 180,E1 18446.035,E2 18446.035} C_VEL
LIN {X 0,Y 376.229,Z 968.637,A -85,B 0,C 180,E1 18442.977,E2 18442.977} C_VEL
LIN {X 0,Y 376.583,Z 964.228,A -85,B 0,C 180,E1 18439.907,E2 18439.907} C_VEL
LIN {X 0,Y 377.292,Z 958.101,A -85,B 0,C 180,E1 18436.825,E2 18436.825} C_VEL
LIN {X 0,Y 378.405,Z 950.566,A -85,B 0,C 180,E1 18433.892,E2 18433.892} C_VEL
LIN {X 0,Y 380.037,Z 941.174,A -85,B 0,C 180,E1 18430.959,E2 18430.959} C_VEL
LIN {X 0,Y 382.132,Z 930.317,A -85,B 0,C 180,E1 18428.188,E2 18428.188} C_VEL
LIN {X 0,Y 384.656,Z 918.023,A -85,B 0,C 180,E1 18425.587,E2 18425.587} C_VEL
LIN {X 0,Y 387.532,Z 904.229,A -85,B 0,C 180,E1 18423.158,E2 18423.158} C_VEL
LIN {X 0,Y 390.687,Z 888.828,A -85,B 0,C 180,E1 18420.904,E2 18420.904} C_VEL
LIN {X 0,Y 393.773,Z 872.989,A -85,B 0,C 180,E1 18418.971,E2 18418.971} C_VEL
LIN {X 0,Y 396.918,Z 855.599,A -85,B 0,C 180,E1 18417.207,E2 18417.207} C_VEL
LIN {X 0,Y 399.909,Z 837.224,A -85,B 0,C 180,E1 18415.68,E2 18415.68} C_VEL
LIN {X 0,Y 402.474,Z 819.036,A -85,B 0,C 180,E1 18414.456,E2 18414.456} C_VEL
LIN {X 0,Y 404.774,Z 799.254,A -85,B 0,C 180,E1 18413.408,E2 18413.408} C_VEL
LIN {X 0,Y 406.586,Z 778.683,A -85,B 0,C 180,E1 18412.602,E2 18412.602} C_VEL
LIN {X 0,Y 407.779,Z 757.689,A -85,B 0,C 180,E1 18412.046,E2 18412.046} C_VEL
LIN {X 0,Y 414.71,Z 548.093,A -85,B 0,C 180,E1 18408.145,E2 18408.145} C_VEL
LIN {X 0,Y 411.94,Z 537.515,A -85,B 0,C 180,E1 18407.55,E2 18407.55} C_VEL
LIN {X 0,Y 400.456,Z 517.235,A -85,B 0,C 180,E1 18405.518,E2 18405.518} C_VEL
LIN {X 0,Y 392.77,Z 504.551,A -85,B 0,C 180,E1 18404.025,E2 18404.025} C_VEL
LIN {X 0,Y 387.608,Z 491.297,A -85,B 0,C 180,E1 18401.128,E2 18401.128} C_VEL
LIN {X 0,Y 386.842,Z 489.971,A -85,B 0,C 180,E1 18400.771,E2 18400.771} C_VEL
LIN {X 0,Y 386.385,Z 489.725,A -85,B 0,C 180,E1 18400.622,E2 18400.622} C_VEL
LIN {X 0,Y 393.185,Z 507.851,A -85,B 0,C 180,E1 18397.245,E2 18397.245} C_VEL
LIN {X 0,Y 399.443,Z 526.471,A -85,B 0,C 180,E1 18394.05,E2 18394.05} C_VEL
LIN {X 0,Y 400.009,Z 529.062,A -85,B 0,C 180,E1 18393.656,E2 18393.656} C_VEL
LIN {X 0,Y 396.482,Z 562.949,A -85,B 0,C 180,E1 18389.706,E2 18389.706} C_VEL
LIN {X 0,Y 393.171,Z 598.612,A -85,B 0,C 180,E1 18385.615,E2 18385.615} C_VEL
LIN {X 0,Y 390.97,Z 626.481,A -85,B 0,C 180,E1 18382.518,E2 18382.518} C_VEL
LIN {X 0,Y 391.523,Z 632.853,A -85,B 0,C 180,E1 18382.291,E2 18382.291} C_VEL
LIN {X 0,Y 385.982,Z 765.005,A -85,B 0,C 180,E1 18378.732,E2 18378.732} C_VEL
LIN {X 0,Y 385.505,Z 782.464,A -85,B 0,C 180,E1 18378.056,E2 18378.056} C_VEL
LIN {X 0,Y 384.764,Z 798.384,A -85,B 0,C 180,E1 18377.154,E2 18377.154} C_VEL
LIN {X 0,Y 383.866,Z 813.532,A -85,B 0,C 180,E1 18376.023,E2 18376.023} C_VEL
LIN {X 0,Y 382.781,Z 828.291,A -85,B 0,C 180,E1 18374.6,E2 18374.6} C_VEL
LIN {X 0,Y 381.707,Z 841.454,A -85,B 0,C 180,E1 18373.019,E2 18373.019} C_VEL
LIN {X 0,Y 380.573,Z 854.471,A -85,B 0,C 180,E1 18371.057,E2 18371.057} C_VEL
LIN {X 0,Y 379.665,Z 864.915,A -85,B 0,C 180,E1 18369.092,E2 18369.092} C_VEL
LIN {X 0,Y 378.888,Z 874.546,A -85,B 0,C 180,E1 18366.82,E2 18366.82} C_VEL
LIN {X 0,Y 378.355,Z 881.959,A -85,B 0,C 180,E1 18364.547,E2 18364.547} C_VEL
LIN {X 0,Y 378.032,Z 887.902,A -85,B 0,C 180,E1 18362.122,E2 18362.122} C_VEL
LIN {X 0,Y 377.927,Z 892.118,A -85,B 0,C 180,E1 18359.545,E2 18359.545} C_VEL
LIN {X 0,Y 378.027,Z 894.318,A -85,B 0,C 180,E1 18357.12,E2 18357.12} C_VEL
LIN {X 0,Y 378.331,Z 894.809,A -85,B 0,C 180,E1 18354.541,E2 18354.541} C_VEL
LIN {X 0,Y 378.845,Z 893.487,A -85,B 0,C 180,E1 18352.112,E2 18352.112} C_VEL
LIN {X 0,Y 379.627,Z 890.496,A -85,B 0,C 180,E1 18349.683,E2 18349.683} C_VEL
LIN {X 0,Y 380.729,Z 885.599,A -85,B 0,C 180,E1 18347.256,E2 18347.256} C_VEL
LIN {X 0,Y 382.063,Z 879.176,A -85,B 0,C 180,E1 18344.985,E2 18344.985} C_VEL
LIN {X 0,Y 383.747,Z 870.699,A -85,B 0,C 180,E1 18342.721,E2 18342.721} C_VEL
LIN {X 0,Y 385.491,Z 861.161,A -85,B 0,C 180,E1 18340.757,E2 18340.757} C_VEL
LIN {X 0,Y 387.4,Z 849.832,A -85,B 0,C 180,E1 18338.897,E2 18338.897} C_VEL
LIN {X 0,Y 389.164,Z 837.894,A -85,B 0,C 180,E1 18337.332,E2 18337.332} C_VEL
LIN {X 0,Y 390.948,Z 823.567,A -85,B 0,C 180,E1 18335.845,E2 18335.845} C_VEL
LIN {X 0,Y 392.292,Z 809.722,A -85,B 0,C 180,E1 18334.728,E2 18334.728} C_VEL
LIN {X 0,Y 393.429,Z 794.667,A -85,B 0,C 180,E1 18333.792,E2 18333.792} C_VEL
LIN {X 0,Y 395.797,Z 765.927,A -85,B 0,C 180,E1 18332.414,E2 18332.414} C_VEL
LIN {X 0,Y 405.905,Z 697.824,A -85,B 0,C 180,E1 18329.517,E2 18329.517} C_VEL
LIN {X 0,Y 410.269,Z 670.023,A -85,B 0,C 180,E1 18328.443,E2 18328.443} C_VEL
LIN {X 0,Y 419.174,Z 655.03,A -85,B 0,C 180,E1 18327.217,E2 18327.217} C_VEL
LIN {X 0,Y 427.421,Z 638.583,A -85,B 0,C 180,E1 18324.497,E2 18324.497} C_VEL
LIN {X 0,Y 435.034,Z 626.914,A -85,B 0,C 180,E1 18322.387,E2 18322.387} C_VEL
LIN {X 0,Y 427.949,Z 638.034,A -85,B 0,C 180,E1 18320.446,E2 18320.446} C_VEL
LIN {X 0,Y 423.41,Z 648.9,A -85,B 0,C 180,E1 18318.468,E2 18318.468} C_VEL
LIN {X 0,Y 421.162,Z 660.586,A -85,B 0,C 180,E1 18316.303,E2 18316.303} C_VEL
LIN {X 0,Y 421.564,Z 671.908,A -85,B 0,C 180,E1 18314.212,E2 18314.212} C_VEL
LIN {X 0,Y 424.501,Z 683.404,A -85,B 0,C 180,E1 18312.103,E2 18312.103} C_VEL
LIN {X 0,Y 429.659,Z 694.708,A -85,B 0,C 180,E1 18310.094,E2 18310.094} C_VEL
LIN {X 0,Y 419.58,Z 713.888,A -85,B 0,C 180,E1 18309.243,E2 18309.243} C_VEL
LIN {X 0,Y 412.796,Z 729.022,A -85,B 0,C 180,E1 18308.474,E2 18308.474} C_VEL
LIN {X 0,Y 409.438,Z 750.562,A -85,B 0,C 180,E1 18308.375,E2 18308.375} C_VEL
LIN {X 0,Y 407.045,Z 773.299,A -85,B 0,C 180,E1 18308.141,E2 18308.141} C_VEL
LIN {X 0,Y 405.759,Z 802.067,A -85,B 0,C 180,E1 18307.571,E2 18307.571} C_VEL
LIN {X 0,Y 404.044,Z 822.767,A -85,B 0,C 180,E1 18306.932,E2 18306.932} C_VEL
LIN {X 0,Y 401.715,Z 843.699,A -85,B 0,C 180,E1 18306.01,E2 18306.01} C_VEL
LIN {X 0,Y 399.007,Z 863.547,A -85,B 0,C 180,E1 18304.844,E2 18304.844} C_VEL
LIN {X 0,Y 396.058,Z 882.31,A -85,B 0,C 180,E1 18303.451,E2 18303.451} C_VEL
LIN {X 0,Y 393.021,Z 899.756,A -85,B 0,C 180,E1 18301.864,E2 18301.864} C_VEL
LIN {X 0,Y 389.775,Z 917.359,A -85,B 0,C 180,E1 18299.922,E2 18299.922} C_VEL
LIN {X 0,Y 386.826,Z 932.852,A -85,B 0,C 180,E1 18297.873,E2 18297.873} C_VEL
LIN {X 0,Y 384.081,Z 947.303,A -85,B 0,C 180,E1 18295.604,E2 18295.604} C_VEL
LIN {X 0,Y 381.514,Z 961.229,A -85,B 0,C 180,E1 18292.986,E2 18292.986} C_VEL
LIN {X 0,Y 379.47,Z 973.538,A -85,B 0,C 180,E1 18290.193,E2 18290.193} C_VEL
LIN {X 0,Y 377.967,Z 983.737,A -85,B 0,C 180,E1 18287.394,E2 18287.394} C_VEL
LIN {X 0,Y 376.941,Z 992.537,A -85,B 0,C 180,E1 18284.439,E2 18284.439} C_VEL
LIN {X 0,Y 376.376,Z 999.843,A -85,B 0,C 180,E1 18281.338,E2 18281.338} C_VEL
LIN {X 0,Y 376.17,Z 1005.088,A -85,B 0,C 180,E1 18278.407,E2 18278.407} C_VEL
LIN {X 0,Y 376.124,Z 1008.693,A -85,B 0,C 180,E1 18275.492,E2 18275.492} C_VEL
LIN {X 0,Y 376.178,Z 1010.754,A -85,B 0,C 180,E1 18272.591,E2 18272.591} C_VEL
LIN {X 0,Y 376.203,Z 1011.369,A -85,B 0,C 180,E1 18269.696,E2 18269.696} C_VEL
LIN {X 0,Y 376.164,Z 1010.469,A -85,B 0,C 180,E1 18266.801,E2 18266.801} C_VEL
LIN {X 0,Y 376.122,Z 1007.964,A -85,B 0,C 180,E1 18263.834,E2 18263.834} C_VEL
LIN {X 0,Y 376.168,Z 1003.842,A -85,B 0,C 180,E1 18260.824,E2 18260.824} C_VEL
LIN {X 0,Y 376.458,Z 998.244,A -85,B 0,C 180,E1 18257.889,E2 18257.889} C_VEL
LIN {X 0,Y 377.151,Z 990.458,A -85,B 0,C 180,E1 18254.785,E2 18254.785} C_VEL
LIN {X 0,Y 378.288,Z 981.098,A -85,B 0,C 180,E1 18251.828,E2 18251.828} C_VEL
LIN {X 0,Y 379.928,Z 970.287,A -85,B 0,C 180,E1 18249.029,E2 18249.029} C_VEL
LIN {X 0,Y 382.081,Z 957.773,A -85,B 0,C 180,E1 18246.334,E2 18246.334} C_VEL
LIN {X 0,Y 384.71,Z 943.557,A -85,B 0,C 180,E1 18243.78,E2 18243.78} C_VEL
LIN {X 0,Y 387.626,Z 928.358,A -85,B 0,C 180,E1 18241.498,E2 18241.498} C_VEL
LIN {X 0,Y 390.694,Z 912.238,A -85,B 0,C 180,E1 18239.47,E2 18239.47} C_VEL
LIN {X 0,Y 393.769,Z 895.337,A -85,B 0,C 180,E1 18237.699,E2 18237.699} C_VEL
LIN {X 0,Y 396.869,Z 876.869,A -85,B 0,C 180,E1 18236.114,E2 18236.114} C_VEL
LIN {X 0,Y 399.573,Z 858.921,A -85,B 0,C 180,E1 18234.864,E2 18234.864} C_VEL
LIN {X 0,Y 402.141,Z 839.16,A -85,B 0,C 180,E1 18233.771,E2 18233.771} C_VEL
LIN {X 0,Y 404.318,Z 818.866,A -85,B 0,C 180,E1 18232.932,E2 18232.932} C_VEL
LIN {X 0,Y 405.902,Z 798.325,A -85,B 0,C 180,E1 18232.335,E2 18232.335} C_VEL
LIN {X 0,Y 407.231,Z 769.107,A -85,B 0,C 180,E1 18231.797,E2 18231.797} C_VEL
LIN {X 0,Y 410.264,Z 741.718,A -85,B 0,C 180,E1 18231.533,E2 18231.533} C_VEL
LIN {X 0,Y 411.074,Z 737.602,A -85,B 0,C 180,E1 18231.49,E2 18231.49} C_VEL
LIN {X 0,Y 424.535,Z 709.405,A -85,B 0,C 180,E1 18229.988,E2 18229.988} C_VEL
LIN {X 0,Y 431.708,Z 696.599,A -85,B 0,C 180,E1 18229.42,E2 18229.42} C_VEL
LIN {X 0,Y 423.739,Z 681.526,A -85,B 0,C 180,E1 18227.375,E2 18227.375} C_VEL
LIN {X 0,Y 418.034,Z 665.649,A -85,B 0,C 180,E1 18225.362,E2 18225.362} C_VEL
LIN {X 0,Y 414.242,Z 648.044,A -85,B 0,C 180,E1 18223.274,E2 18223.274} C_VEL
LIN {X 0,Y 412.534,Z 628.822,A -85,B 0,C 180,E1 18221.15,E2 18221.15} C_VEL
LIN {X 0,Y 413.094,Z 606.835,A -85,B 0,C 180,E1 18218.92,E2 18218.92} C_VEL
LIN {X 0,Y 417.039,Z 575.066,A -85,B 0,C 180,E1 18215.972,E2 18215.972} C_VEL
LIN {X 0,Y 419.98,Z 554.828,A -85,B 0,C 180,E1 18214.101,E2 18214.101} C_VEL
LIN {X 0,Y 410.236,Z 533.701,A -85,B 0,C 180,E1 18210.299,E2 18210.299} C_VEL
LIN {X 0,Y 401.953,Z 516.661,A -85,B 0,C 180,E1 18206.918,E2 18206.918} C_VEL
LIN {X 0,Y 393.775,Z 500.064,A -85,B 0,C 180,E1 18203.335,E2 18203.335} C_VEL
LIN {X 0,Y 386.745,Z 486.525,A -85,B 0,C 180,E1 18200.111,E2 18200.111} C_VEL
LIN {X 0,Y 384.022,Z 481.444,A -85,B 0,C 180,E1 18198.835,E2 18198.835} C_VEL
LIN {X 0,Y 381.723,Z 476.955,A -85,B 0,C 180,E1 18197.688,E2 18197.688} C_VEL
LIN {X 0,Y 379.445,Z 472.541,A -85,B 0,C 180,E1 18196.534,E2 18196.534} C_VEL
LIN {X 0,Y 377.823,Z 469.209,A -85,B 0,C 180,E1 18195.66,E2 18195.66} C_VEL
LIN {X 0,Y 377.691,Z 468.442,A -85,B 0,C 180,E1 18195.506,E2 18195.506} C_VEL
LIN {X 0,Y 377.665,Z 468.443,A -85,B 0,C 180,E1 18191.453,E2 18191.453} C_VEL
LIN {X 0,Y 377.691,Z 468.438,A -85,B 0,C 180,E1 18187.453,E2 18187.453} C_VEL
LIN {X 0,Y 377.649,Z 468.445,A -85,B 0,C 180,E1 18183.491,E2 18183.491} C_VEL
LIN {X 0,Y 377.688,Z 468.441,A -85,B 0,C 180,E1 18179.545,E2 18179.545} C_VEL
LIN {X 0,Y 377.642,Z 468.442,A -85,B 0,C 180,E1 18175.444,E2 18175.444} C_VEL
LIN {X 0,Y 377.681,Z 468.418,A -85,B 0,C 180,E1 18171.474,E2 18171.474} C_VEL
LIN {X 0,Y 377.641,Z 468.424,A -85,B 0,C 180,E1 18167.461,E2 18167.461} C_VEL
LIN {X 0,Y 377.674,Z 468.433,A -85,B 0,C 180,E1 18163.386,E2 18163.386} C_VEL
LIN {X 0,Y 377.65,Z 468.444,A -85,B 0,C 180,E1 18159.382,E2 18159.382} C_VEL
LIN {X 0,Y 377.674,Z 468.444,A -85,B 0,C 180,E1 18155.106,E2 18155.106} C_VEL
LIN {X 0,Y 377.656,Z 468.446,A -85,B 0,C 180,E1 18151.193,E2 18151.193} C_VEL
LIN {X 0,Y 377.67,Z 468.447,A -85,B 0,C 180,E1 18146.95,E2 18146.95} C_VEL
LIN {X 0,Y 377.663,Z 468.439,A -85,B 0,C 180,E1 18143.06,E2 18143.06} C_VEL
LIN {X 0,Y 377.66,Z 468.533,A -85,B 0,C 180,E1 18142.359,E2 18142.359} C_VEL
LIN {X 0,Y 379,Z 471.943,A -85,B 0,C 180,E1 18141.686,E2 18141.686} C_VEL
LIN {X 0,Y 380.234,Z 473.558,A -85,B 0,C 180,E1 18141.256,E2 18141.256} C_VEL
LIN {X 0,Y 381.973,Z 477.184,A -85,B 0,C 180,E1 18140.5,E2 18140.5} C_VEL
LIN {X 0,Y 387.276,Z 487.069,A -85,B 0,C 180,E1 18138.431,E2 18138.431} C_VEL
LIN {X 0,Y 394.832,Z 502.785,A -85,B 0,C 180,E1 18135.557,E2 18135.557} C_VEL
LIN {X 0,Y 406.27,Z 521.417,A -85,B 0,C 180,E1 18133.472,E2 18133.472} C_VEL
LIN {X 0,Y 415.164,Z 537.608,A -85,B 0,C 180,E1 18131.937,E2 18131.937} C_VEL
LIN {X 0,Y 407.477,Z 763.469,A -85,B 0,C 180,E1 18127.727,E2 18127.727} C_VEL
LIN {X 0,Y 406.111,Z 784.038,A -85,B 0,C 180,E1 18127.112,E2 18127.112} C_VEL
LIN {X 0,Y 404.157,Z 804.438,A -85,B 0,C 180,E1 18126.244,E2 18126.244} C_VEL
LIN {X 0,Y 401.854,Z 823.536,A -85,B 0,C 180,E1 18125.169,E2 18125.169} C_VEL
LIN {X 0,Y 399.19,Z 841.928,A -85,B 0,C 180,E1 18123.868,E2 18123.868} C_VEL
LIN {X 0,Y 396.086,Z 860.348,A -85,B 0,C 180,E1 18122.257,E2 18122.257} C_VEL
LIN {X 0,Y 392.914,Z 877.458,A -85,B 0,C 180,E1 18120.423,E2 18120.423} C_VEL
LIN {X 0,Y 389.893,Z 892.538,A -85,B 0,C 180,E1 18118.488,E2 18118.488} C_VEL
LIN {X 0,Y 386.853,Z 907.317,A -85,B 0,C 180,E1 18116.228,E2 18116.228} C_VEL
LIN {X 0,Y 384.091,Z 920.638,A -85,B 0,C 180,E1 18113.796,E2 18113.796} C_VEL
LIN {X 0,Y 381.656,Z 932.732,A -85,B 0,C 180,E1 18111.148,E2 18111.148} C_VEL
LIN {X 0,Y 380.959,Z 936.26,A -85,B 0,C 180,E1 18110.269,E2 18110.269} C_VEL
LIN {X 0,Y 379.282,Z 940.212,A -85,B 0,C 180,E1 18109.293,E2 18109.293} C_VEL
LIN {X 0,Y 371.819,Z 949.549,A -85,B 0,C 180,E1 18106.812,E2 18106.812} C_VEL
LIN {X 0,Y 370.333,Z 952.714,A -85,B 0,C 180,E1 18105.745,E2 18105.745} C_VEL
LIN {X 0,Y 369.213,Z 960.023,A -85,B 0,C 180,E1 18102.67,E2 18102.67} C_VEL
LIN {X 0,Y 368.539,Z 965.723,A -85,B 0,C 180,E1 18099.525,E2 18099.525} C_VEL
LIN {X 0,Y 368.192,Z 969.896,A -85,B 0,C 180,E1 18096.235,E2 18096.235} C_VEL
LIN {X 0,Y 368.059,Z 972.252,A -85,B 0,C 180,E1 18093.114,E2 18093.114} C_VEL
LIN {X 0,Y 368.045,Z 973.076,A -85,B 0,C 180,E1 18089.999,E2 18089.999} C_VEL
LIN {X 0,Y 368.057,Z 972.292,A -85,B 0,C 180,E1 18086.885,E2 18086.885} C_VEL
LIN {X 0,Y 368.187,Z 969.989,A -85,B 0,C 180,E1 18083.763,E2 18083.763} C_VEL
LIN {X 0,Y 368.508,Z 966.111,A -85,B 0,C 180,E1 18080.63,E2 18080.63} C_VEL
LIN {X 0,Y 369.144,Z 960.561,A -85,B 0,C 180,E1 18077.485,E2 18077.485} C_VEL
LIN {X 0,Y 370.265,Z 953.194,A -85,B 0,C 180,E1 18074.333,E2 18074.333} C_VEL
LIN {X 0,Y 371.959,Z 943.789,A -85,B 0,C 180,E1 18071.181,E2 18071.181} C_VEL
LIN {X 0,Y 374.192,Z 932.713,A -85,B 0,C 180,E1 18068.196,E2 18068.196} C_VEL
LIN {X 0,Y 376.762,Z 920.728,A -85,B 0,C 180,E1 18065.542,E2 18065.542} C_VEL
LIN {X 0,Y 379.701,Z 907.342,A -85,B 0,C 180,E1 18063.068,E2 18063.068} C_VEL
LIN {X 0,Y 382.92,Z 892.478,A -85,B 0,C 180,E1 18060.771,E2 18060.771} C_VEL
LIN {X 0,Y 386.358,Z 875.991,A -85,B 0,C 180,E1 18058.655,E2 18058.655} C_VEL
LIN {X 0,Y 389.599,Z 859.155,A -85,B 0,C 180,E1 18056.862,E2 18056.862} C_VEL
LIN {X 0,Y 392.677,Z 841.71,A -85,B 0,C 180,E1 18055.331,E2 18055.331} C_VEL
LIN {X 0,Y 395.507,Z 822.899,A -85,B 0,C 180,E1 18053.996,E2 18053.996} C_VEL
LIN {X 0,Y 397.918,Z 803.479,A -85,B 0,C 180,E1 18052.91,E2 18052.91} C_VEL
LIN {X 0,Y 399.874,Z 783.507,A -85,B 0,C 180,E1 18052.068,E2 18052.068} C_VEL
LIN {X 0,Y 401.289,Z 762.263,A -85,B 0,C 180,E1 18051.442,E2 18051.442} C_VEL
LIN {X 0,Y 408.752,Z 550.058,A -85,B 0,C 180,E1 18047.433,E2 18047.433} C_VEL
LIN {X 0,Y 406.551,Z 541.792,A -85,B 0,C 180,E1 18046.949,E2 18046.949} C_VEL
LIN {X 0,Y 395.547,Z 522.152,A -85,B 0,C 180,E1 18044.935,E2 18044.935} C_VEL
LIN {X 0,Y 385.13,Z 505.198,A -85,B 0,C 180,E1 18042.859,E2 18042.859} C_VEL
LIN {X 0,Y 381.531,Z 496.17,A -85,B 0,C 180,E1 18040.833,E2 18040.833} C_VEL
LIN {X 0,Y 380.51,Z 495.831,A -85,B 0,C 180,E1 18040.53,E2 18040.53} C_VEL
LIN {X 0,Y 386.773,Z 512.716,A -85,B 0,C 180,E1 18037.35,E2 18037.35} C_VEL
LIN {X 0,Y 392.852,Z 530.981,A -85,B 0,C 180,E1 18034.19,E2 18034.19} C_VEL
LIN {X 0,Y 392.377,Z 537.404,A -85,B 0,C 180,E1 18033.396,E2 18033.396} C_VEL
LIN {X 0,Y 388.755,Z 571.233,A -85,B 0,C 180,E1 18029.423,E2 18029.423} C_VEL
LIN {X 0,Y 385.318,Z 607.224,A -85,B 0,C 180,E1 18025.269,E2 18025.269} C_VEL
LIN {X 0,Y 383.698,Z 627.574,A -85,B 0,C 180,E1 18022.993,E2 18022.993} C_VEL
LIN {X 0,Y 384.211,Z 634.043,A -85,B 0,C 180,E1 18022.759,E2 18022.759} C_VEL
LIN {X 0,Y 378.385,Z 764.947,A -85,B 0,C 180,E1 18019.112,E2 18019.112} C_VEL
LIN {X 0,Y 377.881,Z 782.761,A -85,B 0,C 180,E1 18018.418,E2 18018.418} C_VEL
LIN {X 0,Y 377.128,Z 798.693,A -85,B 0,C 180,E1 18017.513,E2 18017.513} C_VEL
LIN {X 0,Y 376.137,Z 814.834,A -85,B 0,C 180,E1 18016.287,E2 18016.287} C_VEL
LIN {X 0,Y 375.009,Z 829.603,A -85,B 0,C 180,E1 18014.831,E2 18014.831} C_VEL
LIN {X 0,Y 373.93,Z 842.405,A -85,B 0,C 180,E1 18013.265,E2 18013.265} C_VEL
LIN {X 0,Y 372.766,Z 855.302,A -85,B 0,C 180,E1 18011.292,E2 18011.292} C_VEL
LIN {X 0,Y 371.819,Z 865.882,A -85,B 0,C 180,E1 18009.28,E2 18009.28} C_VEL
LIN {X 0,Y 371.009,Z 875.557,A -85,B 0,C 180,E1 18006.966,E2 18006.966} C_VEL
LIN {X 0,Y 370.456,Z 883.05,A -85,B 0,C 180,E1 18004.645,E2 18004.645} C_VEL
LIN {X 0,Y 370.123,Z 889.072,A -85,B 0,C 180,E1 18002.168,E2 18002.168} C_VEL
LIN {X 0,Y 370.019,Z 893.364,A -85,B 0,C 180,E1 17999.536,E2 17999.536} C_VEL
LIN {X 0,Y 370.14,Z 895.656,A -85,B 0,C 180,E1 17997.058,E2 17997.058} C_VEL
LIN {X 0,Y 370.477,Z 896.222,A -85,B 0,C 180,E1 17994.425,E2 17994.425} C_VEL
LIN {X 0,Y 371.045,Z 895.002,A -85,B 0,C 180,E1 17991.945,E2 17991.945} C_VEL
LIN {X 0,Y 371.901,Z 892.107,A -85,B 0,C 180,E1 17989.466,E2 17989.466} C_VEL
LIN {X 0,Y 373.095,Z 887.305,A -85,B 0,C 180,E1 17986.991,E2 17986.991} C_VEL
LIN {X 0,Y 374.549,Z 881.047,A -85,B 0,C 180,E1 17984.676,E2 17984.676} C_VEL
LIN {X 0,Y 376.354,Z 872.683,A -85,B 0,C 180,E1 17982.371,E2 17982.371} C_VEL
LIN {X 0,Y 378.227,Z 863.419,A -85,B 0,C 180,E1 17980.383,E2 17980.383} C_VEL
LIN {X 0,Y 380.198,Z 852.797,A -85,B 0,C 180,E1 17978.559,E2 17978.559} C_VEL
LIN {X 0,Y 382.286,Z 840.1,A -85,B 0,C 180,E1 17976.82,E2 17976.82} C_VEL
LIN {X 0,Y 384.207,Z 826.067,A -85,B 0,C 180,E1 17975.312,E2 17975.312} C_VEL
LIN {X 0,Y 385.798,Z 811.802,A -85,B 0,C 180,E1 17974.107,E2 17974.107} C_VEL
LIN {X 0,Y 387.144,Z 795.92,A -85,B 0,C 180,E1 17973.089,E2 17973.089} C_VEL
LIN {X 0,Y 389.896,Z 768.284,A -85,B 0,C 180,E1 17971.679,E2 17971.679} C_VEL
LIN {X 0,Y 398.582,Z 715.086,A -85,B 0,C 180,E1 17969.273,E2 17969.273} C_VEL
LIN {X 0,Y 405.69,Z 673.338,A -85,B 0,C 180,E1 17967.585,E2 17967.585} C_VEL
LIN {X 0,Y 414.738,Z 658.671,A -85,B 0,C 180,E1 17966.408,E2 17966.408} C_VEL
LIN {X 0,Y 421.591,Z 646.027,A -85,B 0,C 180,E1 17964.309,E2 17964.309} C_VEL
LIN {X 0,Y 428.559,Z 635.627,A -85,B 0,C 180,E1 17962.411,E2 17962.411} C_VEL
LIN {X 0,Y 421.607,Z 646.786,A -85,B 0,C 180,E1 17960.362,E2 17960.362} C_VEL
LIN {X 0,Y 417.482,Z 657.345,A -85,B 0,C 180,E1 17958.352,E2 17958.352} C_VEL
LIN {X 0,Y 415.604,Z 668.781,A -85,B 0,C 180,E1 17956.143,E2 17956.143} C_VEL
LIN {X 0,Y 416.275,Z 679.428,A -85,B 0,C 180,E1 17954.096,E2 17954.096} C_VEL
LIN {X 0,Y 419.46,Z 690.688,A -85,B 0,C 180,E1 17951.952,E2 17951.952} C_VEL
LIN {X 0,Y 422.362,Z 697.181,A -85,B 0,C 180,E1 17950.745,E2 17950.745} C_VEL
LIN {X 0,Y 412.548,Z 716.123,A -85,B 0,C 180,E1 17949.871,E2 17949.871} C_VEL
LIN {X 0,Y 406.384,Z 729.538,A -85,B 0,C 180,E1 17949.179,E2 17949.179} C_VEL
LIN {X 0,Y 403.112,Z 751.085,A -85,B 0,C 180,E1 17949.073,E2 17949.073} C_VEL
LIN {X 0,Y 400.765,Z 773.313,A -85,B 0,C 180,E1 17948.844,E2 17948.844} C_VEL
LIN {X 0,Y 399.435,Z 801.595,A -85,B 0,C 180,E1 17948.278,E2 17948.278} C_VEL
LIN {X 0,Y 397.659,Z 822.265,A -85,B 0,C 180,E1 17947.635,E2 17947.635} C_VEL
LIN {X 0,Y 395.22,Z 843.211,A -85,B 0,C 180,E1 17946.705,E2 17946.705} C_VEL
LIN {X 0,Y 392.545,Z 862.034,A -85,B 0,C 180,E1 17945.594,E2 17945.594} C_VEL
LIN {X 0,Y 389.49,Z 880.723,A -85,B 0,C 180,E1 17944.209,E2 17944.209} C_VEL
LIN {X 0,Y 386.252,Z 898.615,A -85,B 0,C 180,E1 17942.578,E2 17942.578} C_VEL
LIN {X 0,Y 383.076,Z 915.049,A -85,B 0,C 180,E1 17940.77,E2 17940.77} C_VEL
LIN {X 0,Y 379.831,Z 931.276,A -85,B 0,C 180,E1 17938.627,E2 17938.627} C_VEL
LIN {X 0,Y 376.758,Z 946.392,A -85,B 0,C 180,E1 17936.234,E2 17936.234} C_VEL
LIN {X 0,Y 373.956,Z 960.728,A -85,B 0,C 180,E1 17933.496,E2 17933.496} C_VEL
LIN {X 0,Y 371.732,Z 973.221,A -85,B 0,C 180,E1 17930.606,E2 17930.606} C_VEL
LIN {X 0,Y 370.127,Z 983.317,A -85,B 0,C 180,E1 17927.774,E2 17927.774} C_VEL
LIN {X 0,Y 369.028,Z 992.119,A -85,B 0,C 180,E1 17924.756,E2 17924.756} C_VEL
LIN {X 0,Y 368.402,Z 999.507,A -85,B 0,C 180,E1 17921.546,E2 17921.546} C_VEL
LIN {X 0,Y 368.172,Z 1004.887,A -85,B 0,C 180,E1 17918.434,E2 17918.434} C_VEL
LIN {X 0,Y 368.129,Z 1008.603,A -85,B 0,C 180,E1 17915.299,E2 17915.299} C_VEL
LIN {X 0,Y 368.193,Z 1010.482,A -85,B 0,C 180,E1 17912.335,E2 17912.335} C_VEL
LIN {X 0,Y 368.21,Z 1010.911,A -85,B 0,C 180,E1 17909.378,E2 17909.378} C_VEL
LIN {X 0,Y 368.166,Z 1009.899,A -85,B 0,C 180,E1 17906.42,E2 17906.42} C_VEL
LIN {X 0,Y 368.131,Z 1007.287,A -85,B 0,C 180,E1 17903.451,E2 17903.451} C_VEL
LIN {X 0,Y 368.204,Z 1002.898,A -85,B 0,C 180,E1 17900.306,E2 17900.306} C_VEL
LIN {X 0,Y 368.569,Z 996.736,A -85,B 0,C 180,E1 17897.148,E2 17897.148} C_VEL
LIN {X 0,Y 369.353,Z 989.123,A -85,B 0,C 180,E1 17894.133,E2 17894.133} C_VEL
LIN {X 0,Y 370.653,Z 979.613,A -85,B 0,C 180,E1 17891.114,E2 17891.114} C_VEL
LIN {X 0,Y 372.594,Z 967.922,A -85,B 0,C 180,E1 17888.1,E2 17888.1} C_VEL
LIN {X 0,Y 374.946,Z 955.287,A -85,B 0,C 180,E1 17885.413,E2 17885.413} C_VEL
LIN {X 0,Y 377.725,Z 941.261,A -85,B 0,C 180,E1 17882.917,E2 17882.917} C_VEL
LIN {X 0,Y 380.872,Z 925.698,A -85,B 0,C 180,E1 17880.601,E2 17880.601} C_VEL
LIN {X 0,Y 384.282,Z 908.458,A -85,B 0,C 180,E1 17878.469,E2 17878.469} C_VEL
LIN {X 0,Y 387.622,Z 890.823,A -85,B 0,C 180,E1 17876.673,E2 17876.673} C_VEL
LIN {X 0,Y 390.685,Z 873.271,A -85,B 0,C 180,E1 17875.201,E2 17875.201} C_VEL
LIN {X 0,Y 393.655,Z 853.993,A -85,B 0,C 180,E1 17873.896,E2 17873.896} C_VEL
LIN {X 0,Y 396.239,Z 834.236,A -85,B 0,C 180,E1 17872.864,E2 17872.864} C_VEL
LIN {X 0,Y 398.318,Z 814.365,A -85,B 0,C 180,E1 17872.095,E2 17872.095} C_VEL
LIN {X 0,Y 399.806,Z 793.197,A -85,B 0,C 180,E1 17871.527,E2 17871.527} C_VEL
LIN {X 0,Y 401.036,Z 768.056,A -85,B 0,C 180,E1 17871.08,E2 17871.08} C_VEL
LIN {X 0,Y 404.12,Z 740.797,A -85,B 0,C 180,E1 17870.824,E2 17870.824} C_VEL
LIN {X 0,Y 405.224,Z 734.755,A -85,B 0,C 180,E1 17870.784,E2 17870.784} C_VEL
LIN {X 0,Y 418.226,Z 707.947,A -85,B 0,C 180,E1 17869.348,E2 17869.348} C_VEL
LIN {X 0,Y 423.489,Z 698.255,A -85,B 0,C 180,E1 17868.892,E2 17868.892} C_VEL
LIN {X 0,Y 415.975,Z 683.147,A -85,B 0,C 180,E1 17866.845,E2 17866.845} C_VEL
LIN {X 0,Y 410.497,Z 666.612,A -85,B 0,C 180,E1 17864.742,E2 17864.742} C_VEL
LIN {X 0,Y 406.95,Z 647.9,A -85,B 0,C 180,E1 17862.517,E2 17862.517} C_VEL
LIN {X 0,Y 405.675,Z 628.686,A -85,B 0,C 180,E1 17860.397,E2 17860.397} C_VEL
LIN {X 0,Y 406.644,Z 606.173,A -85,B 0,C 180,E1 17858.109,E2 17858.109} C_VEL
LIN {X 0,Y 413.406,Z 558.631,A -85,B 0,C 180,E1 17853.67,E2 17853.67} C_VEL
LIN {X 0,Y 403.792,Z 537.697,A -85,B 0,C 180,E1 17849.848,E2 17849.848} C_VEL
LIN {X 0,Y 395.882,Z 521.394,A -85,B 0,C 180,E1 17846.554,E2 17846.554} C_VEL
LIN {X 0,Y 388.038,Z 505.348,A -85,B 0,C 180,E1 17843.058,E2 17843.058} C_VEL
LIN {X 0,Y 380.966,Z 491.739,A -85,B 0,C 180,E1 17839.789,E2 17839.789} C_VEL
LIN {X 0,Y 376.285,Z 482.653,A -85,B 0,C 180,E1 17837.473,E2 17837.473} C_VEL
LIN {X 0,Y 373.861,Z 478.05,A -85,B 0,C 180,E1 17836.239,E2 17836.239} C_VEL
LIN {X 0,Y 371.784,Z 473.835,A -85,B 0,C 180,E1 17835.121,E2 17835.121} C_VEL
LIN {X 0,Y 370.028,Z 470.819,A -85,B 0,C 180,E1 17834.234,E2 17834.234} C_VEL
LIN {X 0,Y 369.731,Z 469.435,A -85,B 0,C 180,E1 17833.874,E2 17833.874} C_VEL
LIN {X 0,Y 369.739,Z 469.43,A -85,B 0,C 180,E1 17829.652,E2 17829.652} C_VEL
LIN {X 0,Y 369.731,Z 469.431,A -85,B 0,C 180,E1 17825.587,E2 17825.587} C_VEL
LIN {X 0,Y 369.746,Z 469.427,A -85,B 0,C 180,E1 17821.239,E2 17821.239} C_VEL
LIN {X 0,Y 369.733,Z 469.431,A -85,B 0,C 180,E1 17817.21,E2 17817.21} C_VEL
LIN {X 0,Y 369.752,Z 469.406,A -85,B 0,C 180,E1 17812.854,E2 17812.854} C_VEL
LIN {X 0,Y 369.739,Z 469.426,A -85,B 0,C 180,E1 17808.772,E2 17808.772} C_VEL
LIN {X 0,Y 369.747,Z 469.43,A -85,B 0,C 180,E1 17804.472,E2 17804.472} C_VEL
LIN {X 0,Y 369.745,Z 469.423,A -85,B 0,C 180,E1 17800.408,E2 17800.408} C_VEL
LIN {X 0,Y 369.743,Z 469.416,A -85,B 0,C 180,E1 17796.239,E2 17796.239} C_VEL
LIN {X 0,Y 369.747,Z 469.417,A -85,B 0,C 180,E1 17792.107,E2 17792.107} C_VEL
LIN {X 0,Y 369.745,Z 469.421,A -85,B 0,C 180,E1 17787.993,E2 17787.993} C_VEL
LIN {X 0,Y 369.754,Z 469.502,A -85,B 0,C 180,E1 17783.835,E2 17783.835} C_VEL
LIN {X 0,Y 370.905,Z 472.71,A -85,B 0,C 180,E1 17783.189,E2 17783.189} C_VEL
LIN {X 0,Y 372.457,Z 474.744,A -85,B 0,C 180,E1 17782.617,E2 17782.617} C_VEL
LIN {X 0,Y 374.607,Z 478.823,A -85,B 0,C 180,E1 17781.693,E2 17781.693} C_VEL
LIN {X 0,Y 380.389,Z 489.872,A -85,B 0,C 180,E1 17779.317,E2 17779.317} C_VEL
LIN {X 0,Y 387.123,Z 503.345,A -85,B 0,C 180,E1 17776.728,E2 17776.728} C_VEL
LIN {X 0,Y 399.795,Z 523.723,A -85,B 0,C 180,E1 17774.309,E2 17774.309} C_VEL
LIN {X 0,Y 409.149,Z 540.624,A -85,B 0,C 180,E1 17772.634,E2 17772.634} C_VEL
LIN {X 0,Y 401.182,Z 763.792,A -85,B 0,C 180,E1 17768.426,E2 17768.426} C_VEL
LIN {X 0,Y 399.763,Z 784.391,A -85,B 0,C 180,E1 17767.804,E2 17767.804} C_VEL
LIN {X 0,Y 397.719,Z 804.891,A -85,B 0,C 180,E1 17766.922,E2 17766.922} C_VEL
LIN {X 0,Y 395.323,Z 823.927,A -85,B 0,C 180,E1 17765.838,E2 17765.838} C_VEL
LIN {X 0,Y 392.543,Z 842.326,A -85,B 0,C 180,E1 17764.522,E2 17764.522} C_VEL
LIN {X 0,Y 389.246,Z 861.035,A -85,B 0,C 180,E1 17762.863,E2 17762.863} C_VEL
LIN {X 0,Y 385.971,Z 877.866,A -85,B 0,C 180,E1 17761.031,E2 17761.031} C_VEL
LIN {X 0,Y 382.685,Z 893.489,A -85,B 0,C 180,E1 17758.99,E2 17758.99} C_VEL
LIN {X 0,Y 379.57,Z 907.855,A -85,B 0,C 180,E1 17756.748,E2 17756.748} C_VEL
LIN {X 0,Y 376.674,Z 921.054,A -85,B 0,C 180,E1 17754.294,E2 17754.294} C_VEL
LIN {X 0,Y 374.127,Z 932.975,A -85,B 0,C 180,E1 17751.641,E2 17751.641} C_VEL
LIN {X 0,Y 372.012,Z 943.486,A -85,B 0,C 180,E1 17748.815,E2 17748.815} C_VEL
LIN {X 0,Y 370.333,Z 952.714,A -85,B 0,C 180,E1 17745.745,E2 17745.745} C_VEL
LIN {X 0,Y 368.903,Z 955.727,A -85,B 0,C 180,E1 17744.658,E2 17744.658} C_VEL
LIN {X 0,Y 361.737,Z 962.764,A -85,B 0,C 180,E1 17741.715,E2 17741.715} C_VEL
LIN {X 0,Y 360.778,Z 964.65,A -85,B 0,C 180,E1 17740.71,E2 17740.71} C_VEL
LIN {X 0,Y 360.304,Z 969.145,A -85,B 0,C 180,E1 17737.493,E2 17737.493} C_VEL
LIN {X 0,Y 360.11,Z 972.006,A -85,B 0,C 180,E1 17734.298,E2 17734.298} C_VEL
LIN {X 0,Y 360.048,Z 973.335,A -85,B 0,C 180,E1 17731.113,E2 17731.113} C_VEL
LIN {X 0,Y 360.055,Z 973.226,A -85,B 0,C 180,E1 17728.09,E2 17728.09} C_VEL
LIN {X 0,Y 360.136,Z 971.527,A -85,B 0,C 180,E1 17724.902,E2 17724.902} C_VEL
LIN {X 0,Y 360.386,Z 968.268,A -85,B 0,C 180,E1 17721.704,E2 17721.704} C_VEL
LIN {X 0,Y 360.964,Z 963.089,A -85,B 0,C 180,E1 17718.333,E2 17718.333} C_VEL
LIN {X 0,Y 361.977,Z 956.357,A -85,B 0,C 180,E1 17715.114,E2 17715.114} C_VEL
LIN {X 0,Y 363.47,Z 948.191,A -85,B 0,C 180,E1 17712.054,E2 17712.054} C_VEL
LIN {X 0,Y 365.575,Z 938.062,A -85,B 0,C 180,E1 17709.004,E2 17709.004} C_VEL
LIN {X 0,Y 368.193,Z 926.37,A -85,B 0,C 180,E1 17706.132,E2 17706.132} C_VEL
LIN {X 0,Y 371.358,Z 912.679,A -85,B 0,C 180,E1 17703.367,E2 17703.367} C_VEL
LIN {X 0,Y 374.772,Z 897.864,A -85,B 0,C 180,E1 17700.898,E2 17700.898} C_VEL
LIN {X 0,Y 378.148,Z 882.627,A -85,B 0,C 180,E1 17698.785,E2 17698.785} C_VEL
LIN {X 0,Y 381.621,Z 865.948,A -85,B 0,C 180,E1 17696.857,E2 17696.857} C_VEL
LIN {X 0,Y 385.027,Z 847.963,A -85,B 0,C 180,E1 17695.146,E2 17695.146} C_VEL
LIN {X 0,Y 388.113,Z 829.469,A -85,B 0,C 180,E1 17693.717,E2 17693.717} C_VEL
LIN {X 0,Y 390.803,Z 810.283,A -85,B 0,C 180,E1 17692.534,E2 17692.534} C_VEL
LIN {X 0,Y 393.09,Z 789.614,A -85,B 0,C 180,E1 17691.563,E2 17691.563} C_VEL
LIN {X 0,Y 394.761,Z 768.519,A -85,B 0,C 180,E1 17690.864,E2 17690.864} C_VEL
LIN {X 0,Y 396.026,Z 738.48,A -85,B 0,C 180,E1 17690.238,E2 17690.238} C_VEL
LIN {X 0,Y 402.81,Z 551.816,A -85,B 0,C 180,E1 17686.688,E2 17686.688} C_VEL
LIN {X 0,Y 401.211,Z 546.043,A -85,B 0,C 180,E1 17686.331,E2 17686.331} C_VEL
LIN {X 0,Y 390.11,Z 526.04,A -85,B 0,C 180,E1 17684.224,E2 17684.224} C_VEL
LIN {X 0,Y 379.607,Z 509.25,A -85,B 0,C 180,E1 17682.093,E2 17682.093} C_VEL
LIN {X 0,Y 377.385,Z 505.65,A -85,B 0,C 180,E1 17681.582,E2 17681.582} C_VEL
LIN {X 0,Y 375.834,Z 502.271,A -85,B 0,C 180,E1 17680.778,E2 17680.778} C_VEL
LIN {X 0,Y 374.646,Z 501.767,A -85,B 0,C 180,E1 17680.46,E2 17680.46} C_VEL
LIN {X 0,Y 381.089,Z 519.6,A -85,B 0,C 180,E1 17677.097,E2 17677.097} C_VEL
LIN {X 0,Y 385.98,Z 534.687,A -85,B 0,C 180,E1 17674.473,E2 17674.473} C_VEL
LIN {X 0,Y 382.188,Z 568.022,A -85,B 0,C 180,E1 17670.5,E2 17670.5} C_VEL
LIN {X 0,Y 378.462,Z 604.877,A -85,B 0,C 180,E1 17666.181,E2 17666.181} C_VEL
LIN {X 0,Y 376.441,Z 628.635,A -85,B 0,C 180,E1 17663.484,E2 17663.484} C_VEL
LIN {X 0,Y 376.931,Z 634.97,A -85,B 0,C 180,E1 17663.25,E2 17663.25} C_VEL
LIN {X 0,Y 370.792,Z 765.308,A -85,B 0,C 180,E1 17659.494,E2 17659.494} C_VEL
LIN {X 0,Y 370.284,Z 782.747,A -85,B 0,C 180,E1 17658.81,E2 17658.81} C_VEL
LIN {X 0,Y 369.507,Z 799.002,A -85,B 0,C 180,E1 17657.886,E2 17657.886} C_VEL
LIN {X 0,Y 368.472,Z 815.282,A -85,B 0,C 180,E1 17656.635,E2 17656.635} C_VEL
LIN {X 0,Y 367.358,Z 829.487,A -85,B 0,C 180,E1 17655.228,E2 17655.228} C_VEL
LIN {X 0,Y 366.141,Z 843.425,A -85,B 0,C 180,E1 17653.503,E2 17653.503} C_VEL
LIN {X 0,Y 364.957,Z 856.06,A -85,B 0,C 180,E1 17651.537,E2 17651.537} C_VEL
LIN {X 0,Y 363.975,Z 866.721,A -85,B 0,C 180,E1 17649.487,E2 17649.487} C_VEL
LIN {X 0,Y 363.125,Z 876.499,A -85,B 0,C 180,E1 17647.118,E2 17647.118} C_VEL
LIN {X 0,Y 362.552,Z 884.106,A -85,B 0,C 180,E1 17644.746,E2 17644.746} C_VEL
LIN {X 0,Y 362.211,Z 890.224,A -85,B 0,C 180,E1 17642.215,E2 17642.215} C_VEL
LIN {X 0,Y 362.113,Z 894.407,A -85,B 0,C 180,E1 17639.684,E2 17639.684} C_VEL
LIN {X 0,Y 362.239,Z 896.91,A -85,B 0,C 180,E1 17637.152,E2 17637.152} C_VEL
LIN {X 0,Y 362.572,Z 897.658,A -85,B 0,C 180,E1 17634.586,E2 17634.586} C_VEL
LIN {X 0,Y 363.164,Z 896.791,A -85,B 0,C 180,E1 17632.088,E2 17632.088} C_VEL
LIN {X 0,Y 364.113,Z 893.945,A -85,B 0,C 180,E1 17629.398,E2 17629.398} C_VEL
LIN {X 0,Y 365.329,Z 889.7,A -85,B 0,C 180,E1 17626.992,E2 17626.992} C_VEL
LIN {X 0,Y 366.935,Z 883.401,A -85,B 0,C 180,E1 17624.512,E2 17624.512} C_VEL
LIN {X 0,Y 368.858,Z 875.384,A -85,B 0,C 180,E1 17622.163,E2 17622.163} C_VEL
LIN {X 0,Y 370.843,Z 866.475,A -85,B 0,C 180,E1 17620.141,E2 17620.141} C_VEL
LIN {X 0,Y 373.135,Z 855.391,A -85,B 0,C 180,E1 17618.132,E2 17618.132} C_VEL
LIN {X 0,Y 375.467,Z 842.427,A -85,B 0,C 180,E1 17616.29,E2 17616.29} C_VEL
LIN {X 0,Y 377.56,Z 828.835,A -85,B 0,C 180,E1 17614.763,E2 17614.763} C_VEL
LIN {X 0,Y 379.412,Z 814.202,A -85,B 0,C 180,E1 17613.469,E2 17613.469} C_VEL
LIN {X 0,Y 380.854,Z 799.659,A -85,B 0,C 180,E1 17612.481,E2 17612.481} C_VEL
LIN {X 0,Y 383.977,Z 772.483,A -85,B 0,C 180,E1 17610.989,E2 17610.989} C_VEL
LIN {X 0,Y 391.245,Z 731.467,A -85,B 0,C 180,E1 17609.006,E2 17609.006} C_VEL
LIN {X 0,Y 400.765,Z 679.663,A -85,B 0,C 180,E1 17606.817,E2 17606.817} C_VEL
LIN {X 0,Y 401.449,Z 676.673,A -85,B 0,C 180,E1 17606.689,E2 17606.689} C_VEL
LIN {X 0,Y 410.454,Z 662.626,A -85,B 0,C 180,E1 17605.588,E2 17605.588} C_VEL
LIN {X 0,Y 411.597,Z 660.755,A -85,B 0,C 180,E1 17605.359,E2 17605.359} C_VEL
LIN {X 0,Y 420.981,Z 645.81,A -85,B 0,C 180,E1 17602.718,E2 17602.718} C_VEL
LIN {X 0,Y 422.078,Z 644.373,A -85,B 0,C 180,E1 17602.403,E2 17602.403} C_VEL
LIN {X 0,Y 415.588,Z 655.051,A -85,B 0,C 180,E1 17600.345,E2 17600.345} C_VEL
LIN {X 0,Y 411.655,Z 665.751,A -85,B 0,C 180,E1 17598.217,E2 17598.217} C_VEL
LIN {X 0,Y 410.154,Z 676.345,A -85,B 0,C 180,E1 17596.085,E2 17596.085} C_VEL
LIN {X 0,Y 411.074,Z 687.034,A -85,B 0,C 180,E1 17593.949,E2 17593.949} C_VEL
LIN {X 0,Y 414.644,Z 698.314,A -85,B 0,C 180,E1 17591.725,E2 17591.725} C_VEL
LIN {X 0,Y 415.205,Z 699.966,A -85,B 0,C 180,E1 17591.425,E2 17591.425} C_VEL
LIN {X 0,Y 405.555,Z 718.838,A -85,B 0,C 180,E1 17590.515,E2 17590.515} C_VEL
LIN {X 0,Y 400.337,Z 729.971,A -85,B 0,C 180,E1 17589.95,E2 17589.95} C_VEL
LIN {X 0,Y 397.928,Z 743.128,A -85,B 0,C 180,E1 17589.859,E2 17589.859} C_VEL
LIN {X 0,Y 394.796,Z 770.136,A -85,B 0,C 180,E1 17589.613,E2 17589.613} C_VEL
LIN {X 0,Y 393.395,Z 798.058,A -85,B 0,C 180,E1 17589.086,E2 17589.086} C_VEL
LIN {X 0,Y 391.616,Z 819.005,A -85,B 0,C 180,E1 17588.459,E2 17588.459} C_VEL
LIN {X 0,Y 389.275,Z 838.772,A -85,B 0,C 180,E1 17587.617,E2 17587.617} C_VEL
LIN {X 0,Y 386.494,Z 858.259,A -85,B 0,C 180,E1 17586.514,E2 17586.514} C_VEL
LIN {X 0,Y 383.36,Z 877.176,A -85,B 0,C 180,E1 17585.152,E2 17585.152} C_VEL
LIN {X 0,Y 379.997,Z 895.257,A -85,B 0,C 180,E1 17583.544,E2 17583.544} C_VEL
LIN {X 0,Y 376.457,Z 912.798,A -85,B 0,C 180,E1 17581.639,E2 17581.639} C_VEL
LIN {X 0,Y 372.87,Z 929.816,A -85,B 0,C 180,E1 17579.389,E2 17579.389} C_VEL
LIN {X 0,Y 369.662,Z 944.631,A -85,B 0,C 180,E1 17577.028,E2 17577.028} C_VEL
LIN {X 0,Y 366.826,Z 958.206,A -85,B 0,C 180,E1 17574.442,E2 17574.442} C_VEL
LIN {X 0,Y 364.502,Z 970.11,A -85,B 0,C 180,E1 17571.736,E2 17571.736} C_VEL
LIN {X 0,Y 362.637,Z 980.794,A -85,B 0,C 180,E1 17568.821,E2 17568.821} C_VEL
LIN {X 0,Y 361.329,Z 990.038,A -85,B 0,C 180,E1 17565.736,E2 17565.736} C_VEL
LIN {X 0,Y 360.534,Z 997.756,A -85,B 0,C 180,E1 17562.494,E2 17562.494} C_VEL
LIN {X 0,Y 360.189,Z 1003.536,A -85,B 0,C 180,E1 17559.266,E2 17559.266} C_VEL
LIN {X 0,Y 360.142,Z 1007.373,A -85,B 0,C 180,E1 17556.217,E2 17556.217} C_VEL
LIN {X 0,Y 360.186,Z 1009.789,A -85,B 0,C 180,E1 17553.024,E2 17553.024} C_VEL
LIN {X 0,Y 360.235,Z 1010.586,A -85,B 0,C 180,E1 17550.001,E2 17550.001} C_VEL
LIN {X 0,Y 360.184,Z 1009.786,A -85,B 0,C 180,E1 17546.977,E2 17546.977} C_VEL
LIN {X 0,Y 360.131,Z 1007.368,A -85,B 0,C 180,E1 17543.785,E2 17543.785} C_VEL
LIN {X 0,Y 360.183,Z 1003.27,A -85,B 0,C 180,E1 17540.574,E2 17540.574} C_VEL
LIN {X 0,Y 360.51,Z 997.715,A -85,B 0,C 180,E1 17537.488,E2 17537.488} C_VEL
LIN {X 0,Y 361.308,Z 990.031,A -85,B 0,C 180,E1 17534.265,E2 17534.265} C_VEL
LIN {X 0,Y 362.608,Z 980.78,A -85,B 0,C 180,E1 17531.18,E2 17531.18} C_VEL
LIN {X 0,Y 364.454,Z 970.091,A -85,B 0,C 180,E1 17528.263,E2 17528.263} C_VEL
LIN {X 0,Y 366.969,Z 957.24,A -85,B 0,C 180,E1 17525.364,E2 17525.364} C_VEL
LIN {X 0,Y 369.808,Z 943.657,A -85,B 0,C 180,E1 17522.812,E2 17522.812} C_VEL
LIN {X 0,Y 372.915,Z 929.209,A -85,B 0,C 180,E1 17520.529,E2 17520.529} C_VEL
LIN {X 0,Y 376.44,Z 912.567,A -85,B 0,C 180,E1 17518.337,E2 17518.337} C_VEL
LIN {X 0,Y 379.928,Z 895.187,A -85,B 0,C 180,E1 17516.451,E2 17516.451} C_VEL
LIN {X 0,Y 383.207,Z 877.535,A -85,B 0,C 180,E1 17514.879,E2 17514.879} C_VEL
LIN {X 0,Y 386.255,Z 859.265,A -85,B 0,C 180,E1 17513.554,E2 17513.554} C_VEL
LIN {X 0,Y 389.065,Z 839.755,A -85,B 0,C 180,E1 17512.432,E2 17512.432} C_VEL
LIN {X 0,Y 391.469,Z 819.568,A -85,B 0,C 180,E1 17511.561,E2 17511.561} C_VEL
LIN {X 0,Y 393.275,Z 798.426,A -85,B 0,C 180,E1 17510.922,E2 17510.922} C_VEL
LIN {X 0,Y 394.712,Z 769.427,A -85,B 0,C 180,E1 17510.373,E2 17510.373} C_VEL
LIN {X 0,Y 397.871,Z 741.019,A -85,B 0,C 180,E1 17510.098,E2 17510.098} C_VEL
LIN {X 0,Y 399.474,Z 731.778,A -85,B 0,C 180,E1 17510.06,E2 17510.06} C_VEL
LIN {X 0,Y 412.413,Z 705.642,A -85,B 0,C 180,E1 17508.651,E2 17508.651} C_VEL
LIN {X 0,Y 415.442,Z 700.189,A -85,B 0,C 180,E1 17508.399,E2 17508.399} C_VEL
LIN {X 0,Y 408.179,Z 684.484,A -85,B 0,C 180,E1 17506.271,E2 17506.271} C_VEL
LIN {X 0,Y 402.987,Z 667.437,A -85,B 0,C 180,E1 17504.103,E2 17504.103} C_VEL
LIN {X 0,Y 399.781,Z 648.26,A -85,B 0,C 180,E1 17501.816,E2 17501.816} C_VEL
LIN {X 0,Y 398.877,Z 628.612,A -85,B 0,C 180,E1 17499.639,E2 17499.639} C_VEL
LIN {X 0,Y 400.26,Z 605.728,A -85,B 0,C 180,E1 17497.299,E2 17497.299} C_VEL
LIN {X 0,Y 406.851,Z 562.477,A -85,B 0,C 180,E1 17493.232,E2 17493.232} C_VEL
LIN {X 0,Y 397.697,Z 542.415,A -85,B 0,C 180,E1 17489.522,E2 17489.522} C_VEL
LIN {X 0,Y 389.78,Z 526.036,A -85,B 0,C 180,E1 17486.181,E2 17486.181} C_VEL
LIN {X 0,Y 382.268,Z 510.589,A -85,B 0,C 180,E1 17482.774,E2 17482.774} C_VEL
LIN {X 0,Y 375.524,Z 497.471,A -85,B 0,C 180,E1 17479.602,E2 17479.602} C_VEL
LIN {X 0,Y 370.524,Z 487.84,A -85,B 0,C 180,E1 17477.106,E2 17477.106} C_VEL
LIN {X 0,Y 368.207,Z 483.418,A -85,B 0,C 180,E1 17475.918,E2 17475.918} C_VEL
LIN {X 0,Y 366.314,Z 479.531,A -85,B 0,C 180,E1 17474.867,E2 17474.867} C_VEL
LIN {X 0,Y 364.341,Z 475.76,A -85,B 0,C 180,E1 17473.813,E2 17473.813} C_VEL
LIN {X 0,Y 362.053,Z 471.751,A -85,B 0,C 180,E1 17472.601,E2 17472.601} C_VEL
LIN {X 0,Y 361.764,Z 470.426,A -85,B 0,C 180,E1 17472.287,E2 17472.287} C_VEL
LIN {X 0,Y 361.806,Z 470.422,A -85,B 0,C 180,E1 17468.102,E2 17468.102} C_VEL
LIN {X 0,Y 361.763,Z 470.426,A -85,B 0,C 180,E1 17463.962,E2 17463.962} C_VEL
LIN {X 0,Y 361.813,Z 470.419,A -85,B 0,C 180,E1 17459.683,E2 17459.683} C_VEL
LIN {X 0,Y 361.763,Z 470.42,A -85,B 0,C 180,E1 17455.561,E2 17455.561} C_VEL
LIN {X 0,Y 361.805,Z 470.394,A -85,B 0,C 180,E1 17451.417,E2 17451.417} C_VEL
LIN {X 0,Y 361.763,Z 470.399,A -85,B 0,C 180,E1 17447.323,E2 17447.323} C_VEL
LIN {X 0,Y 361.804,Z 470.404,A -85,B 0,C 180,E1 17443.132,E2 17443.132} C_VEL
LIN {X 0,Y 361.768,Z 470.419,A -85,B 0,C 180,E1 17438.943,E2 17438.943} C_VEL
LIN {X 0,Y 361.805,Z 470.419,A -85,B 0,C 180,E1 17434.812,E2 17434.812} C_VEL
LIN {X 0,Y 361.77,Z 470.426,A -85,B 0,C 180,E1 17430.712,E2 17430.712} C_VEL
LIN {X 0,Y 361.805,Z 470.416,A -85,B 0,C 180,E1 17426.571,E2 17426.571} C_VEL
LIN {X 0,Y 361.819,Z 470.514,A -85,B 0,C 180,E1 17425.435,E2 17425.435} C_VEL
LIN {X 0,Y 363.158,Z 473.971,A -85,B 0,C 180,E1 17424.677,E2 17424.677} C_VEL
LIN {X 0,Y 364.715,Z 475.961,A -85,B 0,C 180,E1 17424.078,E2 17424.078} C_VEL
LIN {X 0,Y 366.769,Z 479.881,A -85,B 0,C 180,E1 17423.148,E2 17423.148} C_VEL
LIN {X 0,Y 370.68,Z 487.194,A -85,B 0,C 180,E1 17421.457,E2 17421.457} C_VEL
LIN {X 0,Y 375.137,Z 495.535,A -85,B 0,C 180,E1 17419.633,E2 17419.633} C_VEL
LIN {X 0,Y 379.825,Z 504.622,A -85,B 0,C 180,E1 17417.886,E2 17417.886} C_VEL
LIN {X 0,Y 390.658,Z 521.548,A -85,B 0,C 180,E1 17415.701,E2 17415.701} C_VEL
LIN {X 0,Y 401.499,Z 540.46,A -85,B 0,C 180,E1 17413.661,E2 17413.661} C_VEL
LIN {X 0,Y 403.179,Z 544.066,A -85,B 0,C 180,E1 17413.344,E2 17413.344} C_VEL
LIN {X 0,Y 394.94,Z 764.316,A -85,B 0,C 180,E1 17409.142,E2 17409.142} C_VEL
LIN {X 0,Y 393.466,Z 784.854,A -85,B 0,C 180,E1 17408.514,E2 17408.514} C_VEL
LIN {X 0,Y 391.336,Z 805.353,A -85,B 0,C 180,E1 17407.622,E2 17407.622} C_VEL
LIN {X 0,Y 388.848,Z 824.318,A -85,B 0,C 180,E1 17406.531,E2 17406.531} C_VEL
LIN {X 0,Y 385.948,Z 842.724,A -85,B 0,C 180,E1 17405.198,E2 17405.198} C_VEL
LIN {X 0,Y 382.575,Z 861.051,A -85,B 0,C 180,E1 17403.555,E2 17403.555} C_VEL
LIN {X 0,Y 379.074,Z 878.273,A -85,B 0,C 180,E1 17401.66,E2 17401.66} C_VEL
LIN {X 0,Y 375.629,Z 893.9,A -85,B 0,C 180,E1 17399.588,E2 17399.588} C_VEL
LIN {X 0,Y 372.264,Z 908.623,A -85,B 0,C 180,E1 17397.248,E2 17397.248} C_VEL
LIN {X 0,Y 369.112,Z 922.218,A -85,B 0,C 180,E1 17394.654,E2 17394.654} C_VEL
LIN {X 0,Y 366.404,Z 934.186,A -85,B 0,C 180,E1 17391.904,E2 17391.904} C_VEL
LIN {X 0,Y 364.225,Z 944.415,A -85,B 0,C 180,E1 17389.066,E2 17389.066} C_VEL
LIN {X 0,Y 362.427,Z 953.784,A -85,B 0,C 180,E1 17385.849,E2 17385.849} C_VEL
LIN {X 0,Y 361.24,Z 961.122,A -85,B 0,C 180,E1 17382.629,E2 17382.629} C_VEL
LIN {X 0,Y 360.778,Z 964.65,A -85,B 0,C 180,E1 17380.71,E2 17380.71} C_VEL
LIN {X 0,Y 359.59,Z 966.672,A -85,B 0,C 180,E1 17379.533,E2 17379.533} C_VEL
LIN {X 0,Y 354.683,Z 969.933,A -85,B 0,C 180,E1 17377.295,E2 17377.295} C_VEL
LIN {X 0,Y 352.394,Z 971.431,A -85,B 0,C 180,E1 17375.817,E2 17375.817} C_VEL
LIN {X 0,Y 352.161,Z 971.831,A -85,B 0,C 180,E1 17375.277,E2 17375.277} C_VEL
LIN {X 0,Y 352.069,Z 973.6,A -85,B 0,C 180,E1 17371.952,E2 17371.952} C_VEL
LIN {X 0,Y 352.058,Z 973.76,A -85,B 0,C 180,E1 17368.86,E2 17368.86} C_VEL
LIN {X 0,Y 352.123,Z 972.484,A -85,B 0,C 180,E1 17365.602,E2 17365.602} C_VEL
LIN {X 0,Y 352.334,Z 969.676,A -85,B 0,C 180,E1 17362.334,E2 17362.334} C_VEL
LIN {X 0,Y 352.836,Z 965.224,A -85,B 0,C 180,E1 17359.054,E2 17359.054} C_VEL
LIN {X 0,Y 353.768,Z 959.001,A -85,B 0,C 180,E1 17355.765,E2 17355.765} C_VEL
LIN {X 0,Y 355.198,Z 951.276,A -85,B 0,C 180,E1 17352.605,E2 17352.605} C_VEL
LIN {X 0,Y 357.214,Z 941.857,A -85,B 0,C 180,E1 17349.519,E2 17349.519} C_VEL
LIN {X 0,Y 359.773,Z 930.87,A -85,B 0,C 180,E1 17346.582,E2 17346.582} C_VEL
LIN {X 0,Y 362.811,Z 918.427,A -85,B 0,C 180,E1 17343.835,E2 17343.835} C_VEL
LIN {X 0,Y 366.218,Z 904.494,A -85,B 0,C 180,E1 17341.28,E2 17341.28} C_VEL
LIN {X 0,Y 369.93,Z 888.946,A -85,B 0,C 180,E1 17338.919,E2 17338.919} C_VEL
LIN {X 0,Y 373.826,Z 871.573,A -85,B 0,C 180,E1 17336.748,E2 17336.748} C_VEL
LIN {X 0,Y 377.411,Z 853.947,A -85,B 0,C 180,E1 17334.947,E2 17334.947} C_VEL
LIN {X 0,Y 380.573,Z 836.415,A -85,B 0,C 180,E1 17333.481,E2 17333.481} C_VEL
LIN {X 0,Y 383.503,Z 817.652,A -85,B 0,C 180,E1 17332.215,E2 17332.215} C_VEL
LIN {X 0,Y 385.988,Z 798.026,A -85,B 0,C 180,E1 17331.179,E2 17331.179} C_VEL
LIN {X 0,Y 387.903,Z 778.095,A -85,B 0,C 180,E1 17330.396,E2 17330.396} C_VEL
LIN {X 0,Y 389.236,Z 756.727,A -85,B 0,C 180,E1 17329.833,E2 17329.833} C_VEL
LIN {X 0,Y 396.939,Z 553.656,A -85,B 0,C 180,E1 17325.924,E2 17325.924} C_VEL
LIN {X 0,Y 395.844,Z 550.124,A -85,B 0,C 180,E1 17325.681,E2 17325.681} C_VEL
LIN {X 0,Y 385.313,Z 531.054,A -85,B 0,C 180,E1 17323.614,E2 17323.614} C_VEL
LIN {X 0,Y 375.352,Z 514.918,A -85,B 0,C 180,E1 17321.526,E2 17321.526} C_VEL
LIN {X 0,Y 371.677,Z 509.529,A -85,B 0,C 180,E1 17320.72,E2 17320.72} C_VEL
LIN {X 0,Y 369.297,Z 508.871,A -85,B 0,C 180,E1 17320.266,E2 17320.266} C_VEL
LIN {X 0,Y 369.115,Z 508.784,A -85,B 0,C 180,E1 17320.191,E2 17320.191} C_VEL
LIN {X 0,Y 375.575,Z 527.09,A -85,B 0,C 180,E1 17316.742,E2 17316.742} C_VEL
LIN {X 0,Y 378.923,Z 537.861,A -85,B 0,C 180,E1 17314.851,E2 17314.851} C_VEL
LIN {X 0,Y 374.944,Z 571.518,A -85,B 0,C 180,E1 17310.798,E2 17310.798} C_VEL
LIN {X 0,Y 371.046,Z 608.659,A -85,B 0,C 180,E1 17306.4,E2 17306.4} C_VEL
LIN {X 0,Y 369.184,Z 629.643,A -85,B 0,C 180,E1 17303.988,E2 17303.988} C_VEL
LIN {X 0,Y 369.632,Z 636.149,A -85,B 0,C 180,E1 17303.743,E2 17303.743} C_VEL
LIN {X 0,Y 363.215,Z 765.399,A -85,B 0,C 180,E1 17299.896,E2 17299.896} C_VEL
LIN {X 0,Y 362.688,Z 782.757,A -85,B 0,C 180,E1 17299.209,E2 17299.209} C_VEL
LIN {X 0,Y 361.888,Z 799.077,A -85,B 0,C 180,E1 17298.276,E2 17298.276} C_VEL
LIN {X 0,Y 360.804,Z 815.496,A -85,B 0,C 180,E1 17297,E2 17297} C_VEL
LIN {X 0,Y 359.649,Z 829.909,A -85,B 0,C 180,E1 17295.562,E2 17295.562} C_VEL
